FUNCTION_BLOCK "FB303"   // FB303, LAD
TITLE = FB303
{ S7_Optimized_Access := 'TRUE' }
AUTHOR : PRECISE
FAMILY : PRECISE
// SPARGING
// stored: AutoNumber false, MemoryReserve 100, SetENOAutomatically false
   VAR_INPUT
      Enable : Bool;
      Disable : Bool;
      Fault : Bool;
      SecPulse : Bool;
      AlwaysTrue { ExternalVisible := 'False'} : Bool;
      StartConfirmationPopupSel : Bool;   // StartConfirmationPopupSel: 0-NO/1-YES
      EndConfirmationPopupSel : Bool;   // EndConfirmationPopupSel: 0-NO/1-YES
      SpargingModeSel : Int;   // Sparging Mode Selection: 0-DO/1-Time
      SpargingTimebaseSel : Bool;   // Sparging Timebase Selection: 0-sec/1-min
      SpargingLineSel : Bool;   // Sparging LineSelection: 0-THRU GAS FILTER /1-THRU VV
      GasSel : Int;   // Gas Selection - 0-AIR/1-N2
      SetDO : Real := 10.0;   // For Sparging Mode Selection: 0-DO
      SpargingTimeMin : Int := 1;   // For Sparging Mode Selection: 1-Time & Sparging Timebase Selection: 1-min
      SpargingTimeSec : Int := 30;   // For Sparging Mode Selection: 1-Time & Sparging Timebase Selection: 0-sec
      PressuretoOpenVV : Real := 1.0;   // For Sparging LineSelection: 1-THRU VV
      PressuretoCloseVV : Real := 0.5;   // For Sparging LineSelection: 1-THRU VV
      ActualDO : Real;   // For Sparging Mode Selection: 0-DO
      ActualPressure : Real;   // For Sparging LineSelection: 1-THRU VV
      DelaytoOpenGasIn : Int := 3;
   END_VAR
   VAR_OUTPUT
      AirValve : Bool;
      N2Valve : Bool;
      SpargingLineValves : Bool;
      VentValve : Bool;   // For Sparging LineSelection: 1-THRU VV
      StartConfirmationPopup : Bool;   // For Start Confirmation Popup Selection: Yes
      EndConfirmationPopup : Bool;   // For End Confirmation Popup Selection: Yes
      SpargingTimeMinPV : DInt;
      SpargingTimeSecPV : DInt;
      PrintTrigger { ExternalAccessible := 'False'; ExternalVisible := 'False'; ExternalWritable := 'False'} : Bool;
      PrintWord : Int;
      PrintStatus : String[50];
   END_VAR
   VAR_IN_OUT
      Start : Bool;
      Stop : Bool;
      Reset : Bool;
      StartConfirmationAck : Bool;   // For Start Confirmation Popup Selection: Yes
      EndConfirmationAck : Bool;   // For End Confirmation Popup Selection: Yes
      SpareBtn1 : Bool;
      SpareBtn2 : Bool;
      SpareBtn3 : Bool;
      Running : Bool;
      Selected : Bool;
      Paused : Bool;
      StartConfirmationPopupTemp : Bool;   // For Start Confirmation Popup Selection: Yes
      EndConfirmationPopupTemp : Bool;   // For End Confirmation Popup Selection: Yes
      SpargingStarted : Bool;
      SpargingOver : Bool;
      SpargingTimerRunning : Bool;
   END_VAR
   VAR
      ValveOnDelayPV : Int;
      ValveOffDelayPV : Int;
      PrintTriggerTemp : Bool;
      RE1 : Bool;
      RE2 : Bool;
      RE3 : Bool;
      RE4 : Bool;
      RE5 : Bool;
      RE6 : Bool;
      RE7 : Bool;
      SpargingTimer : "FB101";
      PrintTriggerResetTimer { S7_SetPoint := 'True'} : TON_TIME;
      BtnResetTimer { S7_SetPoint := 'True'} : TON_TIME;
   END_VAR
   VAR_TEMP
      STATUS1 : String[40];
      STATUS2 : String[40];
      STATUS3 : String[40];
      STATUS4 : String[40];
      STATUS5 : String[40];
   END_VAR
   VAR_TEMP   // added for the SCL form of the ladder/FBD networks
      _w1 : Bool;
      _w2 : Bool;
      _w3 : Bool;
      _w4 : Bool;
      _w5 : Bool;
   END_VAR
BEGIN

REGION Network 1: Running
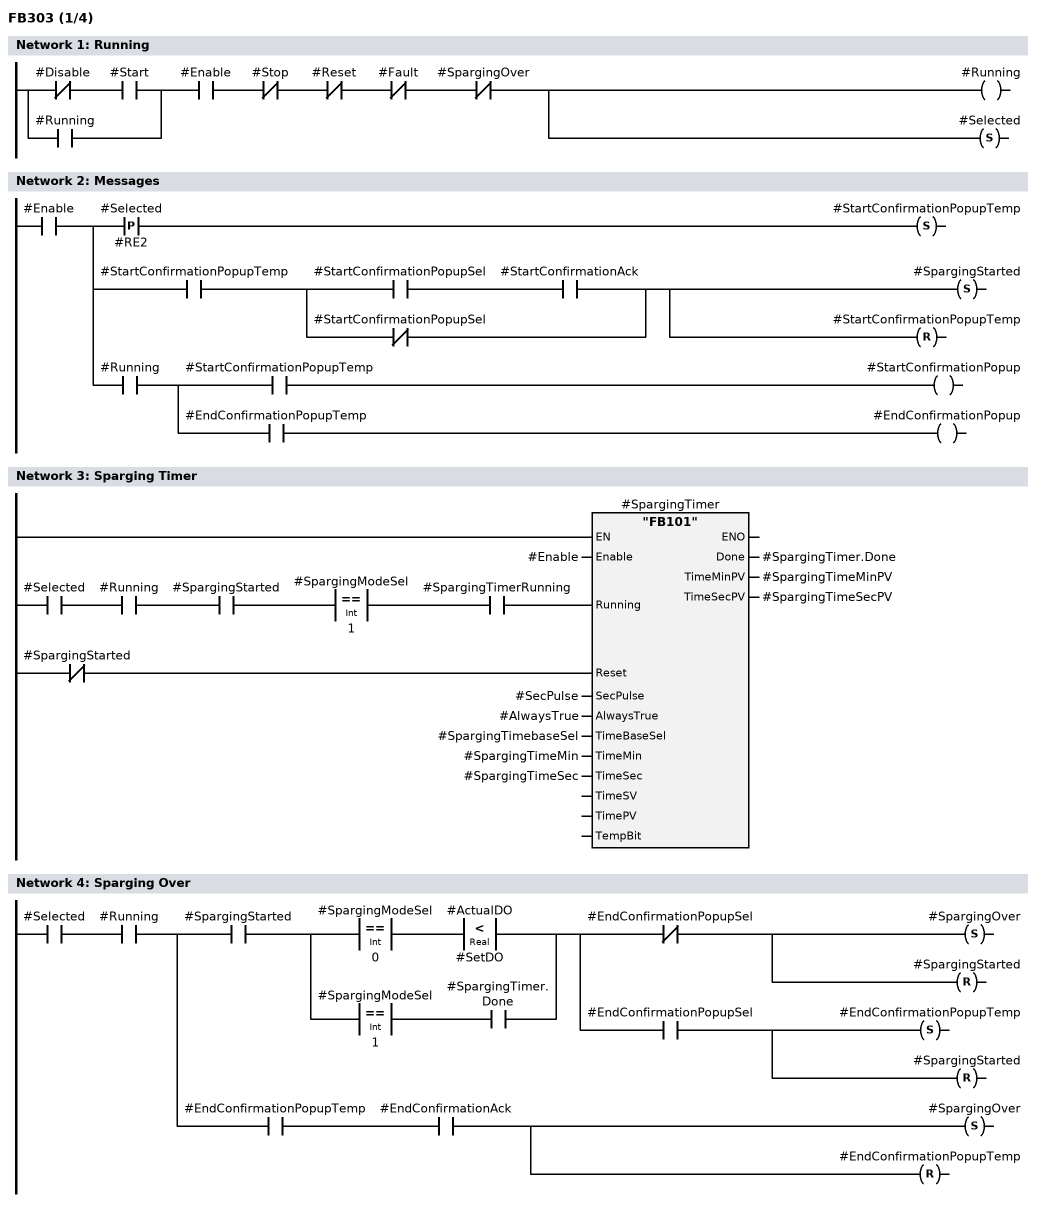
   RUNG wire#powerrail
      I_Contact( #Disable )
      Contact( #Start )
      wire#w1
      Contact( #Enable )
      I_Contact( #Stop )
      I_Contact( #Reset )
      I_Contact( #Fault )
      I_Contact( #SpargingOver )
      wire#w2
      Coil( #Running )
   END_RUNG
   RUNG wire#powerrail
      Contact( #Running )
   END_RUNG wire#w1
   RUNG wire#w2
      S_Coil( #Selected )
   END_RUNG
   // the same network as SCL:
   #Running := ((NOT #Disable AND #Start) OR #Running) AND #Enable AND NOT #Stop AND NOT #Reset AND NOT #Fault AND NOT #SpargingOver;
   IF #Running THEN #Selected := TRUE; END_IF;
END_REGION

REGION Network 2: Messages
   RUNG wire#powerrail
      Contact( #Enable )
      wire#w1
      P_Contact(operand := #Selected, bit := #RE2)
      S_Coil( #StartConfirmationPopupTemp )
   END_RUNG
   RUNG wire#w1
      Contact( #StartConfirmationPopupTemp )
      wire#w2
      Contact( #StartConfirmationPopupSel )
      Contact( #StartConfirmationAck )
      wire#w3
      S_Coil( #SpargingStarted )
   END_RUNG
   RUNG wire#w2
      I_Contact( #StartConfirmationPopupSel )
   END_RUNG wire#w3
   RUNG wire#w3
      R_Coil( #StartConfirmationPopupTemp )
   END_RUNG
   RUNG wire#w1
      Contact( #Running )
      wire#w4
      Contact( #StartConfirmationPopupTemp )
      Coil( #StartConfirmationPopup )
   END_RUNG
   RUNG wire#w4
      Contact( #EndConfirmationPopupTemp )
      Coil( #EndConfirmationPopup )
   END_RUNG
   // the same network as SCL:
   #_w1 := #Enable AND #Selected AND NOT #RE2;   // rising edge of #Selected
   #RE2 := #Selected;
   IF #_w1 THEN #StartConfirmationPopupTemp := TRUE; END_IF;
   IF #Enable AND #StartConfirmationPopupTemp AND ((#StartConfirmationPopupSel AND #StartConfirmationAck) OR NOT #StartConfirmationPopupSel) THEN
       #SpargingStarted := TRUE;
       #StartConfirmationPopupTemp := FALSE;
   END_IF;
   #_w2 := #Enable AND #Running;
   #StartConfirmationPopup := #_w2 AND #StartConfirmationPopupTemp;
   #EndConfirmationPopup := #_w2 AND #EndConfirmationPopupTemp;
END_REGION

REGION Network 3: Sparging Timer
   RUNG wire#powerrail
      #SpargingTimer(Running := wire#w1, Reset := wire#w2, Enable := #Enable, SecPulse := #SecPulse, AlwaysTrue := #AlwaysTrue, TimeBaseSel := #SpargingTimebaseSel, TimeMin := #SpargingTimeMin, TimeSec := #SpargingTimeSec, TimeSV :=, TimePV :=, TempBit :=, Done => #SpargingTimer.Done, TimeMinPV => #SpargingTimeMinPV, TimeSecPV => #SpargingTimeSecPV)
   END_RUNG
   RUNG wire#powerrail
      Contact( #Selected )
      Contact( #Running )
      Contact( #SpargingStarted )
      { S7_Templates := "SrcType := Int" } EQ_Contact(in1 := #SpargingModeSel, in2 := 1)
      Contact( #SpargingTimerRunning )
   END_RUNG wire#w1
   RUNG wire#powerrail
      I_Contact( #SpargingStarted )
   END_RUNG wire#w2
   // the same network as SCL:
   #SpargingTimer(Enable := #Enable,   // "FB101"
                  Running := #Selected AND #Running AND #SpargingStarted AND (#SpargingModeSel = 1) AND #SpargingTimerRunning,
                  Reset := NOT #SpargingStarted,
                  SecPulse := #SecPulse,
                  AlwaysTrue := #AlwaysTrue,
                  TimeBaseSel := #SpargingTimebaseSel,
                  TimeMin := #SpargingTimeMin,
                  TimeSec := #SpargingTimeSec,
                  Done => #SpargingTimer.Done,
                  TimeMinPV => #SpargingTimeMinPV,
                  TimeSecPV => #SpargingTimeSecPV);
END_REGION

REGION Network 4: Sparging Over
   RUNG wire#powerrail
      Contact( #Selected )
      Contact( #Running )
      wire#w1
      Contact( #SpargingStarted )
      wire#w2
      { S7_Templates := "SrcType := Int" } EQ_Contact(in1 := #SpargingModeSel, in2 := 0)
      { S7_Templates := "SrcType := Real" } LT_Contact(in1 := #ActualDO, in2 := #SetDO)
      wire#w3
      I_Contact( #EndConfirmationPopupSel )
      wire#w4
      S_Coil( #SpargingOver )
   END_RUNG
   RUNG wire#w2
      { S7_Templates := "SrcType := Int" } EQ_Contact(in1 := #SpargingModeSel, in2 := 1)
      Contact( #SpargingTimer.Done )
   END_RUNG wire#w3
   RUNG wire#w4
      R_Coil( #SpargingStarted )
   END_RUNG
   RUNG wire#w3
      Contact( #EndConfirmationPopupSel )
      wire#w5
      S_Coil( #EndConfirmationPopupTemp )
   END_RUNG
   RUNG wire#w5
      R_Coil( #SpargingStarted )
   END_RUNG
   RUNG wire#w1
      Contact( #EndConfirmationPopupTemp )
      Contact( #EndConfirmationAck )
      wire#w6
      S_Coil( #SpargingOver )
   END_RUNG
   RUNG wire#w6
      R_Coil( #EndConfirmationPopupTemp )
   END_RUNG
   // the same network as SCL:
   #_w1 := #Selected AND #Running;
   #_w2 := #_w1 AND #SpargingStarted AND (((#SpargingModeSel = 0) AND (#ActualDO < #SetDO)) OR ((#SpargingModeSel = 1) AND #SpargingTimer.Done));
   IF #_w2 AND NOT #EndConfirmationPopupSel THEN
       #SpargingOver := TRUE;
       #SpargingStarted := FALSE;
   END_IF;
   IF #_w2 AND #EndConfirmationPopupSel THEN
       #EndConfirmationPopupTemp := TRUE;
       #SpargingStarted := FALSE;
   END_IF;
   IF #_w1 AND #EndConfirmationPopupTemp AND #EndConfirmationAck THEN
       #SpargingOver := TRUE;
       #EndConfirmationPopupTemp := FALSE;
   END_IF;
END_REGION

REGION Network 5: Output On
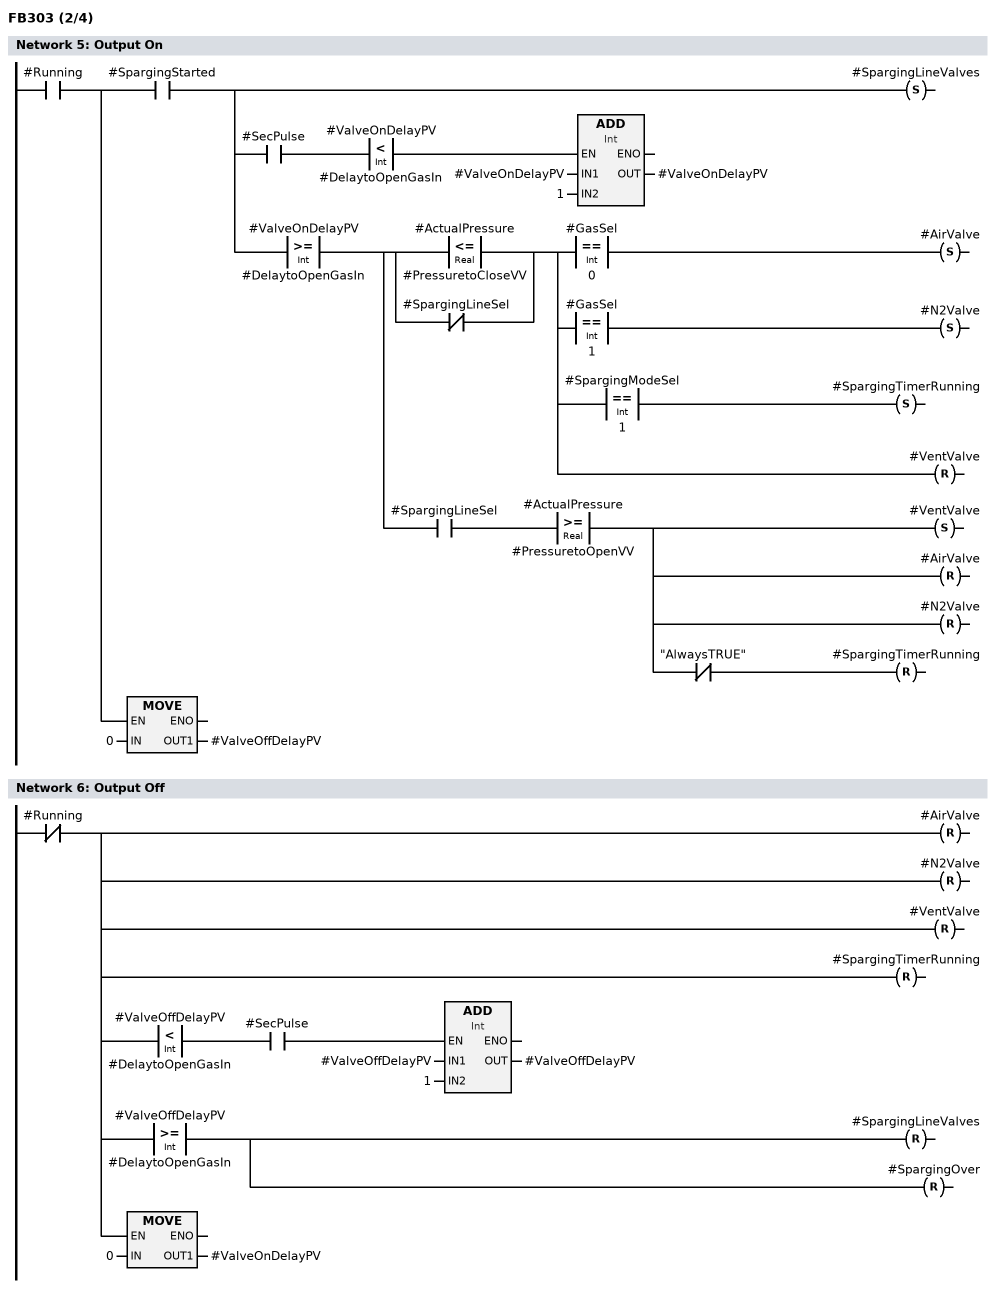
   RUNG wire#powerrail
      Contact( #Running )
      wire#w1
      Contact( #SpargingStarted )
      wire#w2
      S_Coil( #SpargingLineValves )
   END_RUNG
   RUNG wire#w2
      Contact( #SecPulse )
      { S7_Templates := "SrcType := Int" } LT_Contact(in1 := #ValveOnDelayPV, in2 := #DelaytoOpenGasIn)
      { S7_Templates := "SrcType := Int"; S7_GenerateENO := "TRUE" } Add(in1 := #ValveOnDelayPV, in2 := 1, out => #ValveOnDelayPV)
   END_RUNG
   RUNG wire#w2
      { S7_Templates := "SrcType := Int" } GE_Contact(in1 := #ValveOnDelayPV, in2 := #DelaytoOpenGasIn)
      wire#w3
      { S7_Templates := "SrcType := Real" } LE_Contact(in1 := #ActualPressure, in2 := #PressuretoCloseVV)
      wire#w4
      { S7_Templates := "SrcType := Int" } EQ_Contact(in1 := #GasSel, in2 := 0)
      S_Coil( #AirValve )
   END_RUNG
   RUNG wire#w3
      I_Contact( #SpargingLineSel )
   END_RUNG wire#w4
   RUNG wire#w4
      { S7_Templates := "SrcType := Int" } EQ_Contact(in1 := #GasSel, in2 := 1)
      S_Coil( #N2Valve )
   END_RUNG
   RUNG wire#w4
      { S7_Templates := "SrcType := Int" } EQ_Contact(in1 := #SpargingModeSel, in2 := 1)
      S_Coil( #SpargingTimerRunning )
   END_RUNG
   RUNG wire#w4
      R_Coil( #VentValve )
   END_RUNG
   RUNG wire#w3
      Contact( #SpargingLineSel )
      { S7_Templates := "SrcType := Real" } GE_Contact(in1 := #ActualPressure, in2 := #PressuretoOpenVV)
      wire#w5
      S_Coil( #VentValve )
   END_RUNG
   RUNG wire#w5
      R_Coil( #AirValve )
   END_RUNG
   RUNG wire#w5
      R_Coil( #N2Valve )
   END_RUNG
   RUNG wire#w5
      I_Contact( "AlwaysTRUE" )
      R_Coil( #SpargingTimerRunning )
   END_RUNG
   RUNG wire#w1
      { S7_GenerateENO := "TRUE" } Move(in := 0, out1 => #ValveOffDelayPV)
   END_RUNG
   // the same network as SCL:
   #_w1 := #Running AND #SpargingStarted;
   IF #_w1 THEN #SpargingLineValves := TRUE; END_IF;
   IF #_w1 AND #SecPulse AND (#ValveOnDelayPV < #DelaytoOpenGasIn) THEN
       #ValveOnDelayPV := #ValveOnDelayPV + 1;
   END_IF;
   #_w2 := #_w1 AND (#ValveOnDelayPV >= #DelaytoOpenGasIn);
   #_w3 := #_w2 AND ((#ActualPressure <= #PressuretoCloseVV) OR NOT #SpargingLineSel);
   IF #_w3 AND (#GasSel = 0) THEN #AirValve := TRUE; END_IF;
   IF #_w3 AND (#GasSel = 1) THEN #N2Valve := TRUE; END_IF;
   IF #_w3 AND (#SpargingModeSel = 1) THEN #SpargingTimerRunning := TRUE; END_IF;
   IF #_w3 THEN #VentValve := FALSE; END_IF;
   #_w4 := #_w2 AND #SpargingLineSel AND (#ActualPressure >= #PressuretoOpenVV);
   IF #_w4 THEN
       #VentValve := TRUE;
       #AirValve := FALSE;
       #N2Valve := FALSE;
   END_IF;
   IF #_w4 AND NOT "AlwaysTRUE" THEN #SpargingTimerRunning := FALSE; END_IF;
   IF #Running THEN #ValveOffDelayPV := 0; END_IF;
END_REGION

REGION Network 6: Output Off
   RUNG wire#powerrail
      I_Contact( #Running )
      wire#w1
      R_Coil( #AirValve )
   END_RUNG
   RUNG wire#w1
      R_Coil( #N2Valve )
   END_RUNG
   RUNG wire#w1
      R_Coil( #VentValve )
   END_RUNG
   RUNG wire#w1
      R_Coil( #SpargingTimerRunning )
   END_RUNG
   RUNG wire#w1
      { S7_Templates := "SrcType := Int" } LT_Contact(in1 := #ValveOffDelayPV, in2 := #DelaytoOpenGasIn)
      Contact( #SecPulse )
      { S7_Templates := "SrcType := Int"; S7_GenerateENO := "TRUE" } Add(in1 := #ValveOffDelayPV, in2 := 1, out => #ValveOffDelayPV)
   END_RUNG
   RUNG wire#w1
      { S7_Templates := "SrcType := Int" } GE_Contact(in1 := #ValveOffDelayPV, in2 := #DelaytoOpenGasIn)
      wire#w2
      R_Coil( #SpargingLineValves )
   END_RUNG
   RUNG wire#w2
      R_Coil( #SpargingOver )
   END_RUNG
   RUNG wire#w1
      { S7_GenerateENO := "TRUE" } Move(in := 0, out1 => #ValveOnDelayPV)
   END_RUNG
   // the same network as SCL:
   IF NOT #Running THEN
       #AirValve := FALSE;
       #N2Valve := FALSE;
       #VentValve := FALSE;
       #SpargingTimerRunning := FALSE;
   END_IF;
   IF NOT #Running AND (#ValveOffDelayPV < #DelaytoOpenGasIn) AND #SecPulse THEN
       #ValveOffDelayPV := #ValveOffDelayPV + 1;
   END_IF;
   IF NOT #Running AND (#ValveOffDelayPV >= #DelaytoOpenGasIn) THEN
       #SpargingLineValves := FALSE;
       #SpargingOver := FALSE;
   END_IF;
   IF NOT #Running THEN #ValveOnDelayPV := 0; END_IF;
END_REGION

REGION Network 7: Event Status
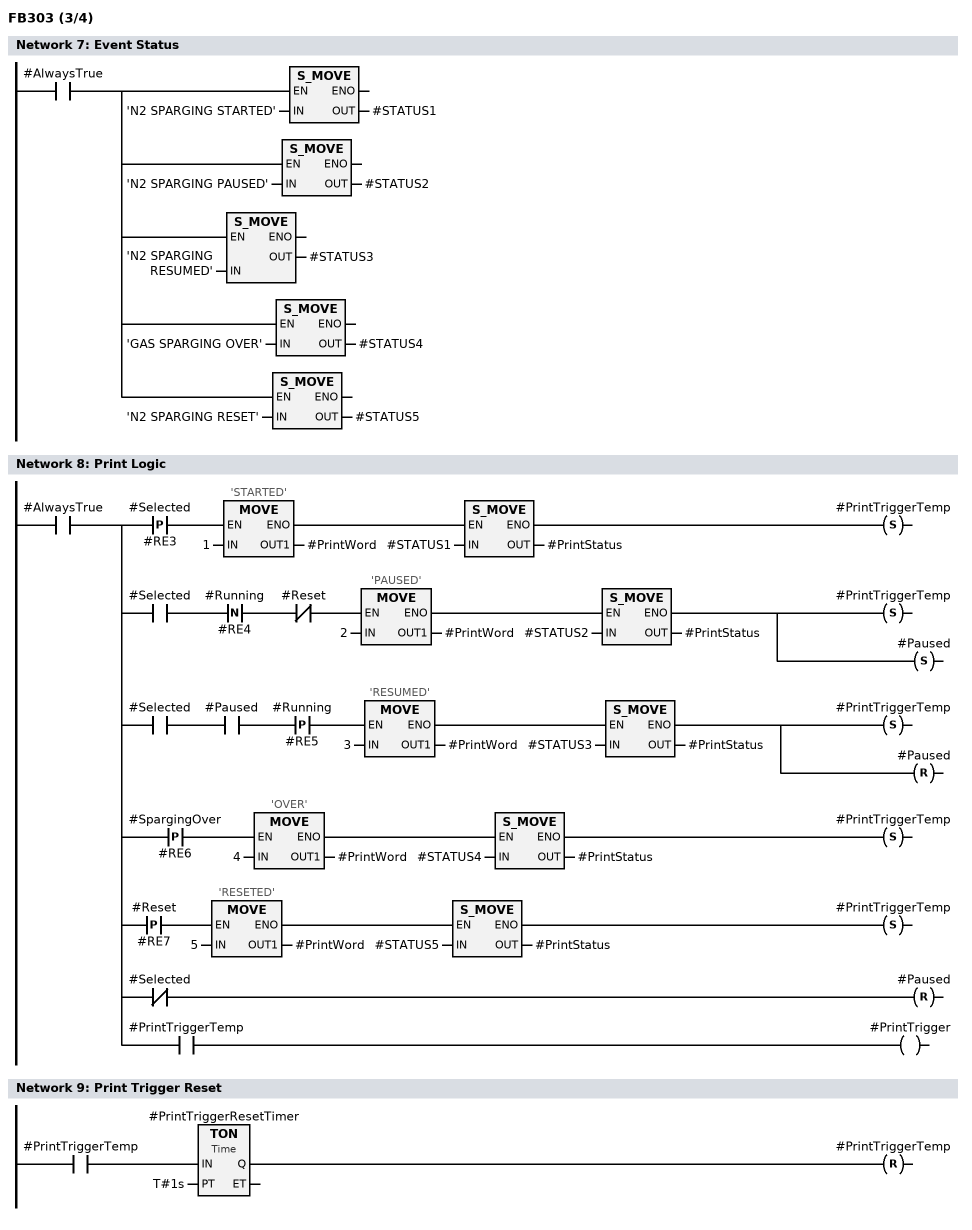
   RUNG wire#powerrail
      Contact( #AlwaysTrue )
      wire#w1
      S_Move(in := 'N2 SPARGING STARTED', out => #STATUS1)
   END_RUNG
   RUNG wire#w1
      S_Move(in := 'N2 SPARGING PAUSED', out => #STATUS2)
   END_RUNG
   RUNG wire#w1
      S_Move(in := 'N2 SPARGING RESUMED', out => #STATUS3)
   END_RUNG
   RUNG wire#w1
      S_Move(in := 'GAS SPARGING OVER', out => #STATUS4)
   END_RUNG
   RUNG wire#w1
      S_Move(in := 'N2 SPARGING RESET', out => #STATUS5)
   END_RUNG
   // the same network as SCL:
   IF #AlwaysTrue THEN
       #STATUS1 := 'N2 SPARGING STARTED';
       #STATUS2 := 'N2 SPARGING PAUSED';
       #STATUS3 := 'N2 SPARGING RESUMED';
       #STATUS4 := 'GAS SPARGING OVER';
       #STATUS5 := 'N2 SPARGING RESET';
   END_IF;
END_REGION

REGION Network 8: Print Logic
   RUNG wire#powerrail
      Contact( #AlwaysTrue )
      wire#w1
      P_Contact(operand := #Selected, bit := #RE3)
      { S7_GenerateENO := "TRUE" } Move(in := 1, out1 => #PrintWord)   // 'STARTED'
      S_Move(in := #STATUS1, out => #PrintStatus)
      S_Coil( #PrintTriggerTemp )
   END_RUNG
   RUNG wire#w1
      Contact( #Selected )
      N_Contact(operand := #Running, bit := #RE4)
      I_Contact( #Reset )
      { S7_GenerateENO := "TRUE" } Move(in := 2, out1 => #PrintWord)   // 'PAUSED'
      S_Move(in := #STATUS2, out => #PrintStatus)
      wire#w2
      S_Coil( #PrintTriggerTemp )
   END_RUNG
   RUNG wire#w2
      S_Coil( #Paused )
   END_RUNG
   RUNG wire#w1
      Contact( #Selected )
      Contact( #Paused )
      P_Contact(operand := #Running, bit := #RE5)
      { S7_GenerateENO := "TRUE" } Move(in := 3, out1 => #PrintWord)   // 'RESUMED'
      S_Move(in := #STATUS3, out => #PrintStatus)
      wire#w3
      S_Coil( #PrintTriggerTemp )
   END_RUNG
   RUNG wire#w3
      R_Coil( #Paused )
   END_RUNG
   RUNG wire#w1
      P_Contact(operand := #SpargingOver, bit := #RE6)
      { S7_GenerateENO := "TRUE" } Move(in := 4, out1 => #PrintWord)   // 'OVER'
      S_Move(in := #STATUS4, out => #PrintStatus)
      S_Coil( #PrintTriggerTemp )
   END_RUNG
   RUNG wire#w1
      P_Contact(operand := #Reset, bit := #RE7)
      { S7_GenerateENO := "TRUE" } Move(in := 5, out1 => #PrintWord)   // 'RESETED'
      S_Move(in := #STATUS5, out => #PrintStatus)
      S_Coil( #PrintTriggerTemp )
   END_RUNG
   RUNG wire#w1
      I_Contact( #Selected )
      R_Coil( #Paused )
   END_RUNG
   RUNG wire#w1
      Contact( #PrintTriggerTemp )
      Coil( #PrintTrigger )
   END_RUNG
   // the same network as SCL:
   // ENO of a box is taken as its EN; it also drops when the box reports an error
   #_w1 := #AlwaysTrue AND #Selected AND NOT #RE3;   // rising edge of #Selected
   #RE3 := #Selected;
   IF #_w1 THEN
       #PrintWord := 1;   // 'STARTED'
       #PrintStatus := #STATUS1;
       #PrintTriggerTemp := TRUE;
   END_IF;
   #_w2 := #AlwaysTrue AND #Selected AND NOT #Running AND #RE4;   // falling edge of #Running
   #RE4 := #Running;
   IF #_w2 AND NOT #Reset THEN
       #PrintWord := 2;   // 'PAUSED'
       #PrintStatus := #STATUS2;
       #PrintTriggerTemp := TRUE;
       #Paused := TRUE;
   END_IF;
   #_w3 := #AlwaysTrue AND #Selected AND #Paused AND #Running AND NOT #RE5;   // rising edge of #Running
   #RE5 := #Running;
   IF #_w3 THEN
       #PrintWord := 3;   // 'RESUMED'
       #PrintStatus := #STATUS3;
       #PrintTriggerTemp := TRUE;
       #Paused := FALSE;
   END_IF;
   #_w4 := #AlwaysTrue AND #SpargingOver AND NOT #RE6;   // rising edge of #SpargingOver
   #RE6 := #SpargingOver;
   IF #_w4 THEN
       #PrintWord := 4;   // 'OVER'
       #PrintStatus := #STATUS4;
       #PrintTriggerTemp := TRUE;
   END_IF;
   #_w5 := #AlwaysTrue AND #Reset AND NOT #RE7;   // rising edge of #Reset
   #RE7 := #Reset;
   IF #_w5 THEN
       #PrintWord := 5;   // 'RESETED'
       #PrintStatus := #STATUS5;
       #PrintTriggerTemp := TRUE;
   END_IF;
   IF #AlwaysTrue AND NOT #Selected THEN #Paused := FALSE; END_IF;
   #PrintTrigger := #AlwaysTrue AND #PrintTriggerTemp;
END_REGION

REGION Network 9: Print Trigger Reset
   RUNG wire#powerrail
      Contact( #PrintTriggerTemp )
      { S7_Templates := "time_type := Time" } #PrintTriggerResetTimer.TON(pt := T#1s, et =>)
      R_Coil( #PrintTriggerTemp )
   END_RUNG
   // the same network as SCL:
   #PrintTriggerResetTimer(IN := #PrintTriggerTemp, PT := T#1s);   // TON
   IF #PrintTriggerResetTimer.Q THEN #PrintTriggerTemp := FALSE; END_IF;
END_REGION

REGION Network 10: Button Reset
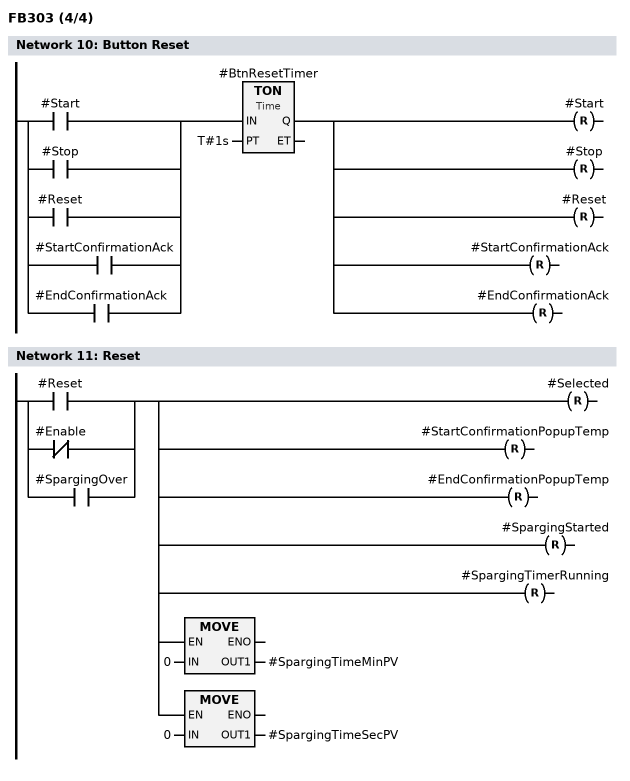
   RUNG wire#powerrail
      Contact( #Start )
      wire#w1
      { S7_Templates := "time_type := Time" } #BtnResetTimer.TON(pt := T#1s, et =>)
      wire#w2
      R_Coil( #Start )
   END_RUNG
   RUNG wire#powerrail
      Contact( #Stop )
   END_RUNG wire#w1
   RUNG wire#powerrail
      Contact( #Reset )
   END_RUNG wire#w1
   RUNG wire#powerrail
      Contact( #StartConfirmationAck )
   END_RUNG wire#w1
   RUNG wire#powerrail
      Contact( #EndConfirmationAck )
   END_RUNG wire#w1
   RUNG wire#w2
      R_Coil( #Stop )
   END_RUNG
   RUNG wire#w2
      R_Coil( #Reset )
   END_RUNG
   RUNG wire#w2
      R_Coil( #StartConfirmationAck )
   END_RUNG
   RUNG wire#w2
      R_Coil( #EndConfirmationAck )
   END_RUNG
   // the same network as SCL:
   #BtnResetTimer(IN := #Start OR #Stop OR #Reset OR #StartConfirmationAck OR #EndConfirmationAck, PT := T#1s);   // TON
   IF #BtnResetTimer.Q THEN
       #Start := FALSE;
       #Stop := FALSE;
       #Reset := FALSE;
       #StartConfirmationAck := FALSE;
       #EndConfirmationAck := FALSE;
   END_IF;
END_REGION

REGION Network 11: Reset
   RUNG wire#powerrail
      Contact( #Reset )
      wire#w1
      R_Coil( #Selected )
   END_RUNG
   RUNG wire#powerrail
      I_Contact( #Enable )
   END_RUNG wire#w1
   RUNG wire#powerrail
      Contact( #SpargingOver )
   END_RUNG wire#w1
   RUNG wire#w1
      R_Coil( #StartConfirmationPopupTemp )
   END_RUNG
   RUNG wire#w1
      R_Coil( #EndConfirmationPopupTemp )
   END_RUNG
   RUNG wire#w1
      R_Coil( #SpargingStarted )
   END_RUNG
   RUNG wire#w1
      R_Coil( #SpargingTimerRunning )
   END_RUNG
   RUNG wire#w1
      { S7_GenerateENO := "TRUE" } Move(in := 0, out1 => #SpargingTimeMinPV)
   END_RUNG
   RUNG wire#w1
      { S7_GenerateENO := "TRUE" } Move(in := 0, out1 => #SpargingTimeSecPV)
   END_RUNG
   // the same network as SCL:
   IF #Reset OR NOT #Enable OR #SpargingOver THEN
       #Selected := FALSE;
       #StartConfirmationPopupTemp := FALSE;
       #EndConfirmationPopupTemp := FALSE;
       #SpargingStarted := FALSE;
       #SpargingTimerRunning := FALSE;
       #SpargingTimeMinPV := 0;
       #SpargingTimeSecPV := 0;
   END_IF;
END_REGION
END_FUNCTION_BLOCK

FUNCTION_BLOCK "FB304"   // FB304, LAD
TITLE = FB304
{ S7_Optimized_Access := 'TRUE' }
AUTHOR : PRECISE
FAMILY : PRECISE
// BLANKETING
// stored: AutoNumber false, MemoryReserve 100, SetENOAutomatically false
   VAR_INPUT
      Enable : Bool;
      Disable : Bool;
      Fault : Bool;
      SecPulse : Bool;
      AlwaysTrue : Bool;
      StartConfirmationPopupSel : Bool;   // StartConfirmationPopupSel: 0-NO/1-YES
      EndConfirmationPopupSel : Bool;   // EndConfirmationPopupSel: 0-NO/1-YES
      BlanketingModeSel : Int;   // Blanketing Mode Selection: 0-Pressure/1-Pressure+Time
      BlanketingTimebaseSel : Bool;   // Blanketing Timebase Selection: 0-sec/1-min
      GasSel : Int;   // Gas Selection - 0-AIR/1-N2
      SetPressure : Real := 1.0;   // For Blanketing Mode Selection: 0-Pressure
      BlanketingTimeMin : Int := 1;   // For Blanketing Mode Selection: 1-Pressure+Time & Blanketing Timebase Selection: 1-min
      BlanketingTimeSec : Int := 30;   // For Blanketing Mode Selection: 1-Pressure+Time & Blanketing Timebase Selection: 0-sec
      ActualPressure : Real;   // For Sparging LineSelection: 1-THRU VV
      DelaytoOpenGasIn : Int := 3;
      PressureTol : Real := 0.3;
   END_VAR
   VAR_OUTPUT
      AirValve : Bool;
      N2Valve : Bool;
      BlanketingLineValves : Bool;
      StartConfirmationPopup : Bool;   // For Start Confirmation Popup Selection: Yes
      EndConfirmationPopup : Bool;   // For End Confirmation Popup Selection: Yes
      BlanketingTimeMinPV : DInt;
      BlanketingTimeSecPV : DInt;
      PrintTrigger : Bool;
      PrintWord : Int;
      PrintStatus : String[50];
   END_VAR
   VAR_IN_OUT
      Start : Bool;
      Stop : Bool;
      Reset : Bool;
      StartConfirmationAck : Bool;   // For Start Confirmation Popup Selection: Yes
      EndConfirmationAck : Bool;   // For End Confirmation Popup Selection: Yes
      SpareBtn1 : Bool;
      SpareBtn2 : Bool;
      SpareBtn3 : Bool;
      Running : Bool;
      Selected : Bool;
      Paused : Bool;
      StartConfirmationPopupTemp : Bool;   // For Start Confirmation Popup Selection: Yes
      EndConfirmationPopupTemp : Bool;   // For End Confirmation Popup Selection: Yes
      BlanketingStarted : Bool;
      BlanketingOver : Bool;
      BlanketingTimerRunning : Bool;
      PressureTolNeg : Real;
   END_VAR
   VAR
      ValveOnDelayPV : Int;
      ValveOffDelayPV : Int;
      PrintTriggerTemp : Bool;
      RE1 : Bool;
      RE2 : Bool;
      RE3 : Bool;
      RE4 : Bool;
      RE5 : Bool;
      RE6 : Bool;
      RE7 : Bool;
      BlanketingTimer { S7_SetPoint := 'True'} : "FB101";
      PrintTriggerResetTimer { S7_SetPoint := 'True'} : TON_TIME;
      BtnResetTimer { S7_SetPoint := 'True'} : TON_TIME;
   END_VAR
   VAR_TEMP
      STATUS1 : String[40];
      STATUS2 : String[40];
      STATUS3 : String[40];
      STATUS4 : String[40];
      STATUS5 : String[40];
   END_VAR
   VAR_TEMP   // added for the SCL form of the ladder/FBD networks
      _w1 : Bool;
      _w2 : Bool;
      _w3 : Bool;
      _w4 : Bool;
      _w5 : Bool;
   END_VAR
BEGIN

REGION Network 1: Running
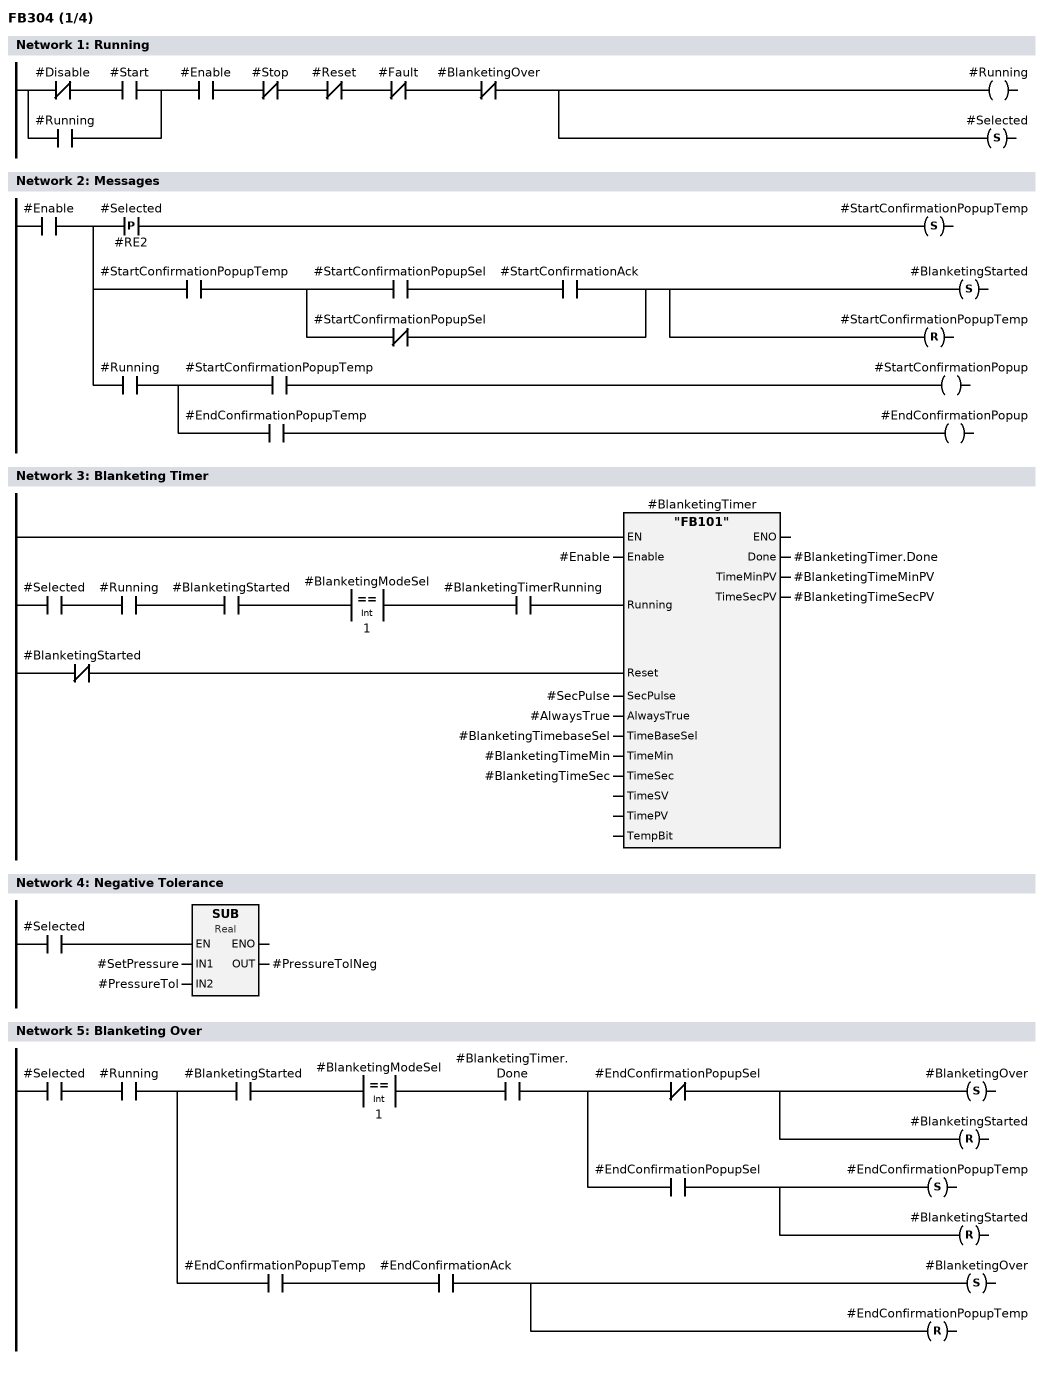
   RUNG wire#powerrail
      I_Contact( #Disable )
      Contact( #Start )
      wire#w1
      Contact( #Enable )
      I_Contact( #Stop )
      I_Contact( #Reset )
      I_Contact( #Fault )
      I_Contact( #BlanketingOver )
      wire#w2
      Coil( #Running )
   END_RUNG
   RUNG wire#powerrail
      Contact( #Running )
   END_RUNG wire#w1
   RUNG wire#w2
      S_Coil( #Selected )
   END_RUNG
   // the same network as SCL:
   #Running := ((NOT #Disable AND #Start) OR #Running) AND #Enable AND NOT #Stop AND NOT #Reset AND NOT #Fault AND NOT #BlanketingOver;
   IF #Running THEN #Selected := TRUE; END_IF;
END_REGION

REGION Network 2: Messages
   RUNG wire#powerrail
      Contact( #Enable )
      wire#w1
      P_Contact(operand := #Selected, bit := #RE2)
      S_Coil( #StartConfirmationPopupTemp )
   END_RUNG
   RUNG wire#w1
      Contact( #StartConfirmationPopupTemp )
      wire#w2
      Contact( #StartConfirmationPopupSel )
      Contact( #StartConfirmationAck )
      wire#w3
      S_Coil( #BlanketingStarted )
   END_RUNG
   RUNG wire#w2
      I_Contact( #StartConfirmationPopupSel )
   END_RUNG wire#w3
   RUNG wire#w3
      R_Coil( #StartConfirmationPopupTemp )
   END_RUNG
   RUNG wire#w1
      Contact( #Running )
      wire#w4
      Contact( #StartConfirmationPopupTemp )
      Coil( #StartConfirmationPopup )
   END_RUNG
   RUNG wire#w4
      Contact( #EndConfirmationPopupTemp )
      Coil( #EndConfirmationPopup )
   END_RUNG
   // the same network as SCL:
   #_w1 := #Enable AND #Selected AND NOT #RE2;   // rising edge of #Selected
   #RE2 := #Selected;
   IF #_w1 THEN #StartConfirmationPopupTemp := TRUE; END_IF;
   IF #Enable AND #StartConfirmationPopupTemp AND ((#StartConfirmationPopupSel AND #StartConfirmationAck) OR NOT #StartConfirmationPopupSel) THEN
       #BlanketingStarted := TRUE;
       #StartConfirmationPopupTemp := FALSE;
   END_IF;
   #_w2 := #Enable AND #Running;
   #StartConfirmationPopup := #_w2 AND #StartConfirmationPopupTemp;
   #EndConfirmationPopup := #_w2 AND #EndConfirmationPopupTemp;
END_REGION

REGION Network 3: Blanketing Timer
   RUNG wire#powerrail
      #BlanketingTimer(Running := wire#w1, Reset := wire#w2, Enable := #Enable, SecPulse := #SecPulse, AlwaysTrue := #AlwaysTrue, TimeBaseSel := #BlanketingTimebaseSel, TimeMin := #BlanketingTimeMin, TimeSec := #BlanketingTimeSec, TimeSV :=, TimePV :=, TempBit :=, Done => #BlanketingTimer.Done, TimeMinPV => #BlanketingTimeMinPV, TimeSecPV => #BlanketingTimeSecPV)
   END_RUNG
   RUNG wire#powerrail
      Contact( #Selected )
      Contact( #Running )
      Contact( #BlanketingStarted )
      { S7_Templates := "SrcType := Int" } EQ_Contact(in1 := #BlanketingModeSel, in2 := 1)
      Contact( #BlanketingTimerRunning )
   END_RUNG wire#w1
   RUNG wire#powerrail
      I_Contact( #BlanketingStarted )
   END_RUNG wire#w2
   // the same network as SCL:
   #BlanketingTimer(Enable := #Enable,   // "FB101"
                    Running := #Selected AND #Running AND #BlanketingStarted AND (#BlanketingModeSel = 1) AND #BlanketingTimerRunning,
                    Reset := NOT #BlanketingStarted,
                    SecPulse := #SecPulse,
                    AlwaysTrue := #AlwaysTrue,
                    TimeBaseSel := #BlanketingTimebaseSel,
                    TimeMin := #BlanketingTimeMin,
                    TimeSec := #BlanketingTimeSec,
                    Done => #BlanketingTimer.Done,
                    TimeMinPV => #BlanketingTimeMinPV,
                    TimeSecPV => #BlanketingTimeSecPV);
END_REGION

REGION Network 4: Negative Tolerance
   RUNG wire#powerrail
      Contact( #Selected )
      { S7_Templates := "SrcType := Real"; S7_GenerateENO := "TRUE" } Sub(in1 := #SetPressure, in2 := #PressureTol, out => #PressureTolNeg)
   END_RUNG
   // the same network as SCL:
   IF #Selected THEN #PressureTolNeg := #SetPressure - #PressureTol; END_IF;
END_REGION

REGION Network 5: Blanketing Over
   RUNG wire#powerrail
      Contact( #Selected )
      Contact( #Running )
      wire#w1
      Contact( #BlanketingStarted )
      { S7_Templates := "SrcType := Int" } EQ_Contact(in1 := #BlanketingModeSel, in2 := 1)
      Contact( #BlanketingTimer.Done )
      wire#w2
      I_Contact( #EndConfirmationPopupSel )
      wire#w3
      S_Coil( #BlanketingOver )
   END_RUNG
   RUNG wire#w3
      R_Coil( #BlanketingStarted )
   END_RUNG
   RUNG wire#w2
      Contact( #EndConfirmationPopupSel )
      wire#w4
      S_Coil( #EndConfirmationPopupTemp )
   END_RUNG
   RUNG wire#w4
      R_Coil( #BlanketingStarted )
   END_RUNG
   RUNG wire#w1
      Contact( #EndConfirmationPopupTemp )
      Contact( #EndConfirmationAck )
      wire#w5
      S_Coil( #BlanketingOver )
   END_RUNG
   RUNG wire#w5
      R_Coil( #EndConfirmationPopupTemp )
   END_RUNG
   // the same network as SCL:
   #_w1 := #Selected AND #Running;
   #_w2 := #_w1 AND #BlanketingStarted AND (#BlanketingModeSel = 1) AND #BlanketingTimer.Done;
   IF #_w2 AND NOT #EndConfirmationPopupSel THEN
       #BlanketingOver := TRUE;
       #BlanketingStarted := FALSE;
   END_IF;
   IF #_w2 AND #EndConfirmationPopupSel THEN
       #EndConfirmationPopupTemp := TRUE;
       #BlanketingStarted := FALSE;
   END_IF;
   IF #_w1 AND #EndConfirmationPopupTemp AND #EndConfirmationAck THEN
       #BlanketingOver := TRUE;
       #EndConfirmationPopupTemp := FALSE;
   END_IF;
END_REGION

REGION Network 6: Output On
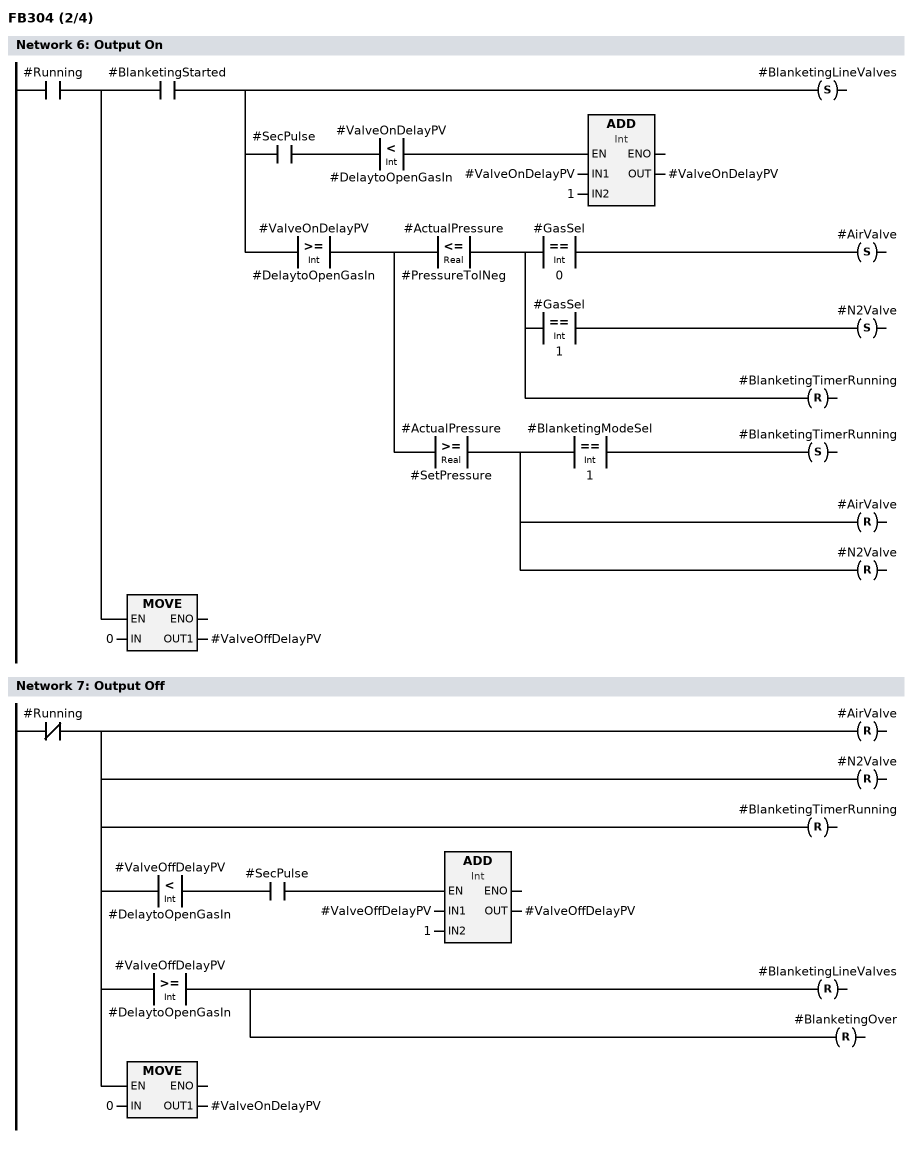
   RUNG wire#powerrail
      Contact( #Running )
      wire#w1
      Contact( #BlanketingStarted )
      wire#w2
      S_Coil( #BlanketingLineValves )
   END_RUNG
   RUNG wire#w2
      Contact( #SecPulse )
      { S7_Templates := "SrcType := Int" } LT_Contact(in1 := #ValveOnDelayPV, in2 := #DelaytoOpenGasIn)
      { S7_Templates := "SrcType := Int"; S7_GenerateENO := "TRUE" } Add(in1 := #ValveOnDelayPV, in2 := 1, out => #ValveOnDelayPV)
   END_RUNG
   RUNG wire#w2
      { S7_Templates := "SrcType := Int" } GE_Contact(in1 := #ValveOnDelayPV, in2 := #DelaytoOpenGasIn)
      wire#w3
      { S7_Templates := "SrcType := Real" } LE_Contact(in1 := #ActualPressure, in2 := #PressureTolNeg)
      wire#w4
      { S7_Templates := "SrcType := Int" } EQ_Contact(in1 := #GasSel, in2 := 0)
      S_Coil( #AirValve )
   END_RUNG
   RUNG wire#w4
      { S7_Templates := "SrcType := Int" } EQ_Contact(in1 := #GasSel, in2 := 1)
      S_Coil( #N2Valve )
   END_RUNG
   RUNG wire#w4
      R_Coil( #BlanketingTimerRunning )
   END_RUNG
   RUNG wire#w3
      { S7_Templates := "SrcType := Real" } GE_Contact(in1 := #ActualPressure, in2 := #SetPressure)
      wire#w5
      { S7_Templates := "SrcType := Int" } EQ_Contact(in1 := #BlanketingModeSel, in2 := 1)
      S_Coil( #BlanketingTimerRunning )
   END_RUNG
   RUNG wire#w5
      R_Coil( #AirValve )
   END_RUNG
   RUNG wire#w5
      R_Coil( #N2Valve )
   END_RUNG
   RUNG wire#w1
      { S7_GenerateENO := "TRUE" } Move(in := 0, out1 => #ValveOffDelayPV)
   END_RUNG
   // the same network as SCL:
   #_w1 := #Running AND #BlanketingStarted;
   IF #_w1 THEN #BlanketingLineValves := TRUE; END_IF;
   IF #_w1 AND #SecPulse AND (#ValveOnDelayPV < #DelaytoOpenGasIn) THEN
       #ValveOnDelayPV := #ValveOnDelayPV + 1;
   END_IF;
   #_w2 := #_w1 AND (#ValveOnDelayPV >= #DelaytoOpenGasIn);
   #_w3 := #_w2 AND (#ActualPressure <= #PressureTolNeg);
   IF #_w3 AND (#GasSel = 0) THEN #AirValve := TRUE; END_IF;
   IF #_w3 AND (#GasSel = 1) THEN #N2Valve := TRUE; END_IF;
   IF #_w3 THEN #BlanketingTimerRunning := FALSE; END_IF;
   #_w4 := #_w2 AND (#ActualPressure >= #SetPressure);
   IF #_w4 AND (#BlanketingModeSel = 1) THEN #BlanketingTimerRunning := TRUE; END_IF;
   IF #_w4 THEN
       #AirValve := FALSE;
       #N2Valve := FALSE;
   END_IF;
   IF #Running THEN #ValveOffDelayPV := 0; END_IF;
END_REGION

REGION Network 7: Output Off
   RUNG wire#powerrail
      I_Contact( #Running )
      wire#w1
      R_Coil( #AirValve )
   END_RUNG
   RUNG wire#w1
      R_Coil( #N2Valve )
   END_RUNG
   RUNG wire#w1
      R_Coil( #BlanketingTimerRunning )
   END_RUNG
   RUNG wire#w1
      { S7_Templates := "SrcType := Int" } LT_Contact(in1 := #ValveOffDelayPV, in2 := #DelaytoOpenGasIn)
      Contact( #SecPulse )
      { S7_Templates := "SrcType := Int"; S7_GenerateENO := "TRUE" } Add(in1 := #ValveOffDelayPV, in2 := 1, out => #ValveOffDelayPV)
   END_RUNG
   RUNG wire#w1
      { S7_Templates := "SrcType := Int" } GE_Contact(in1 := #ValveOffDelayPV, in2 := #DelaytoOpenGasIn)
      wire#w2
      R_Coil( #BlanketingLineValves )
   END_RUNG
   RUNG wire#w2
      R_Coil( #BlanketingOver )
   END_RUNG
   RUNG wire#w1
      { S7_GenerateENO := "TRUE" } Move(in := 0, out1 => #ValveOnDelayPV)
   END_RUNG
   // the same network as SCL:
   IF NOT #Running THEN
       #AirValve := FALSE;
       #N2Valve := FALSE;
       #BlanketingTimerRunning := FALSE;
   END_IF;
   IF NOT #Running AND (#ValveOffDelayPV < #DelaytoOpenGasIn) AND #SecPulse THEN
       #ValveOffDelayPV := #ValveOffDelayPV + 1;
   END_IF;
   IF NOT #Running AND (#ValveOffDelayPV >= #DelaytoOpenGasIn) THEN
       #BlanketingLineValves := FALSE;
       #BlanketingOver := FALSE;
   END_IF;
   IF NOT #Running THEN #ValveOnDelayPV := 0; END_IF;
END_REGION

REGION Network 8: Event Status
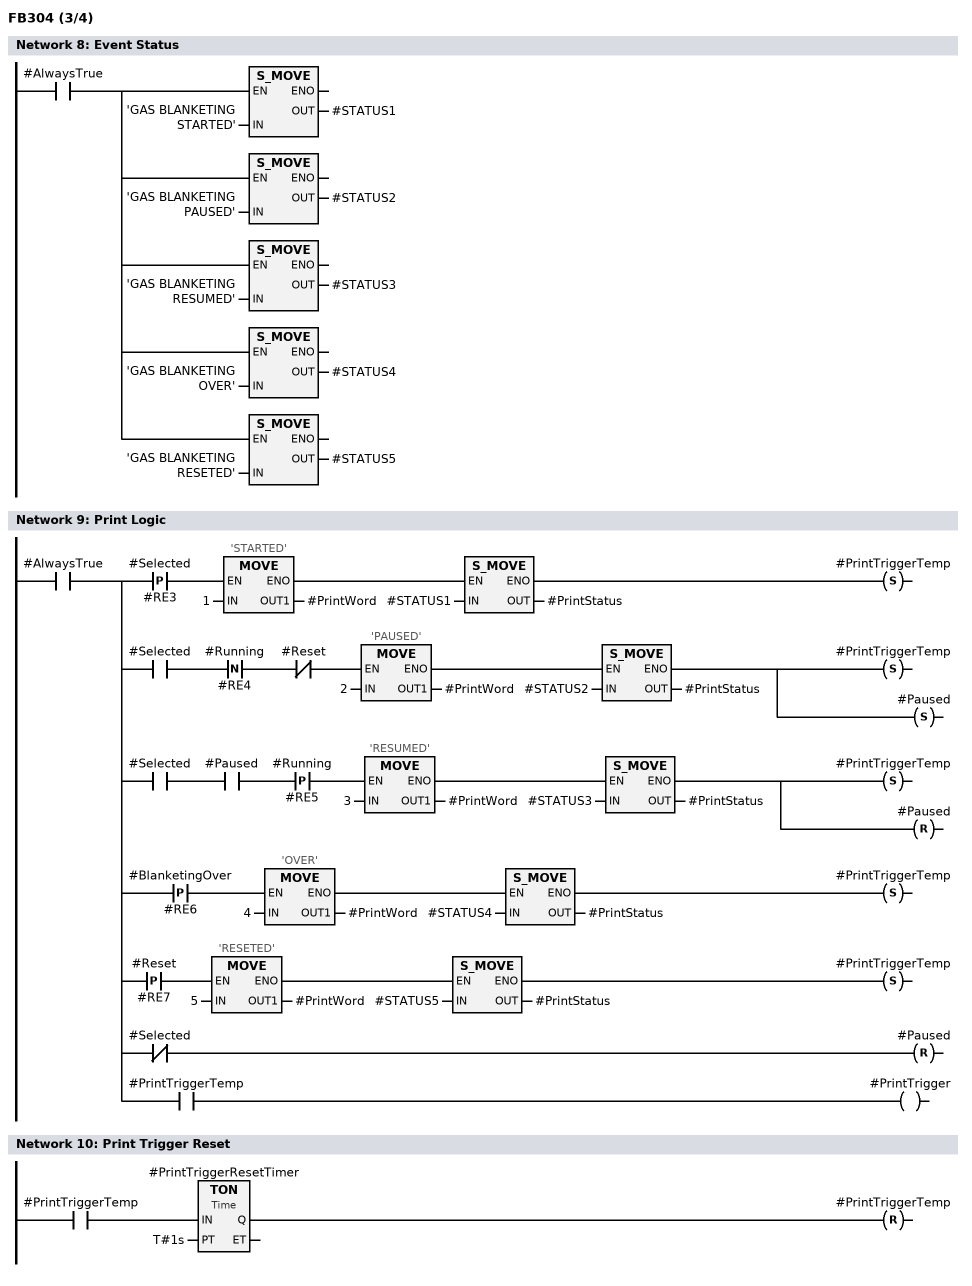
   RUNG wire#powerrail
      Contact( #AlwaysTrue )
      wire#w1
      S_Move(in := 'GAS BLANKETING STARTED', out => #STATUS1)
   END_RUNG
   RUNG wire#w1
      S_Move(in := 'GAS BLANKETING PAUSED', out => #STATUS2)
   END_RUNG
   RUNG wire#w1
      S_Move(in := 'GAS BLANKETING RESUMED', out => #STATUS3)
   END_RUNG
   RUNG wire#w1
      S_Move(in := 'GAS BLANKETING OVER', out => #STATUS4)
   END_RUNG
   RUNG wire#w1
      S_Move(in := 'GAS BLANKETING RESETED', out => #STATUS5)
   END_RUNG
   // the same network as SCL:
   IF #AlwaysTrue THEN
       #STATUS1 := 'GAS BLANKETING STARTED';
       #STATUS2 := 'GAS BLANKETING PAUSED';
       #STATUS3 := 'GAS BLANKETING RESUMED';
       #STATUS4 := 'GAS BLANKETING OVER';
       #STATUS5 := 'GAS BLANKETING RESETED';
   END_IF;
END_REGION

REGION Network 9: Print Logic
   RUNG wire#powerrail
      Contact( #AlwaysTrue )
      wire#w1
      P_Contact(operand := #Selected, bit := #RE3)
      { S7_GenerateENO := "TRUE" } Move(in := 1, out1 => #PrintWord)   // 'STARTED'
      S_Move(in := #STATUS1, out => #PrintStatus)
      S_Coil( #PrintTriggerTemp )
   END_RUNG
   RUNG wire#w1
      Contact( #Selected )
      N_Contact(operand := #Running, bit := #RE4)
      I_Contact( #Reset )
      { S7_GenerateENO := "TRUE" } Move(in := 2, out1 => #PrintWord)   // 'PAUSED'
      S_Move(in := #STATUS2, out => #PrintStatus)
      wire#w2
      S_Coil( #PrintTriggerTemp )
   END_RUNG
   RUNG wire#w2
      S_Coil( #Paused )
   END_RUNG
   RUNG wire#w1
      Contact( #Selected )
      Contact( #Paused )
      P_Contact(operand := #Running, bit := #RE5)
      { S7_GenerateENO := "TRUE" } Move(in := 3, out1 => #PrintWord)   // 'RESUMED'
      S_Move(in := #STATUS3, out => #PrintStatus)
      wire#w3
      S_Coil( #PrintTriggerTemp )
   END_RUNG
   RUNG wire#w3
      R_Coil( #Paused )
   END_RUNG
   RUNG wire#w1
      P_Contact(operand := #BlanketingOver, bit := #RE6)
      { S7_GenerateENO := "TRUE" } Move(in := 4, out1 => #PrintWord)   // 'OVER'
      S_Move(in := #STATUS4, out => #PrintStatus)
      S_Coil( #PrintTriggerTemp )
   END_RUNG
   RUNG wire#w1
      P_Contact(operand := #Reset, bit := #RE7)
      { S7_GenerateENO := "TRUE" } Move(in := 5, out1 => #PrintWord)   // 'RESETED'
      S_Move(in := #STATUS5, out => #PrintStatus)
      S_Coil( #PrintTriggerTemp )
   END_RUNG
   RUNG wire#w1
      I_Contact( #Selected )
      R_Coil( #Paused )
   END_RUNG
   RUNG wire#w1
      Contact( #PrintTriggerTemp )
      Coil( #PrintTrigger )
   END_RUNG
   // the same network as SCL:
   // ENO of a box is taken as its EN; it also drops when the box reports an error
   #_w1 := #AlwaysTrue AND #Selected AND NOT #RE3;   // rising edge of #Selected
   #RE3 := #Selected;
   IF #_w1 THEN
       #PrintWord := 1;   // 'STARTED'
       #PrintStatus := #STATUS1;
       #PrintTriggerTemp := TRUE;
   END_IF;
   #_w2 := #AlwaysTrue AND #Selected AND NOT #Running AND #RE4;   // falling edge of #Running
   #RE4 := #Running;
   IF #_w2 AND NOT #Reset THEN
       #PrintWord := 2;   // 'PAUSED'
       #PrintStatus := #STATUS2;
       #PrintTriggerTemp := TRUE;
       #Paused := TRUE;
   END_IF;
   #_w3 := #AlwaysTrue AND #Selected AND #Paused AND #Running AND NOT #RE5;   // rising edge of #Running
   #RE5 := #Running;
   IF #_w3 THEN
       #PrintWord := 3;   // 'RESUMED'
       #PrintStatus := #STATUS3;
       #PrintTriggerTemp := TRUE;
       #Paused := FALSE;
   END_IF;
   #_w4 := #AlwaysTrue AND #BlanketingOver AND NOT #RE6;   // rising edge of #BlanketingOver
   #RE6 := #BlanketingOver;
   IF #_w4 THEN
       #PrintWord := 4;   // 'OVER'
       #PrintStatus := #STATUS4;
       #PrintTriggerTemp := TRUE;
   END_IF;
   #_w5 := #AlwaysTrue AND #Reset AND NOT #RE7;   // rising edge of #Reset
   #RE7 := #Reset;
   IF #_w5 THEN
       #PrintWord := 5;   // 'RESETED'
       #PrintStatus := #STATUS5;
       #PrintTriggerTemp := TRUE;
   END_IF;
   IF #AlwaysTrue AND NOT #Selected THEN #Paused := FALSE; END_IF;
   #PrintTrigger := #AlwaysTrue AND #PrintTriggerTemp;
END_REGION

REGION Network 10: Print Trigger Reset
   RUNG wire#powerrail
      Contact( #PrintTriggerTemp )
      { S7_Templates := "time_type := Time" } #PrintTriggerResetTimer.TON(pt := T#1s, et =>)
      R_Coil( #PrintTriggerTemp )
   END_RUNG
   // the same network as SCL:
   #PrintTriggerResetTimer(IN := #PrintTriggerTemp, PT := T#1s);   // TON
   IF #PrintTriggerResetTimer.Q THEN #PrintTriggerTemp := FALSE; END_IF;
END_REGION

REGION Network 11: Button Reset
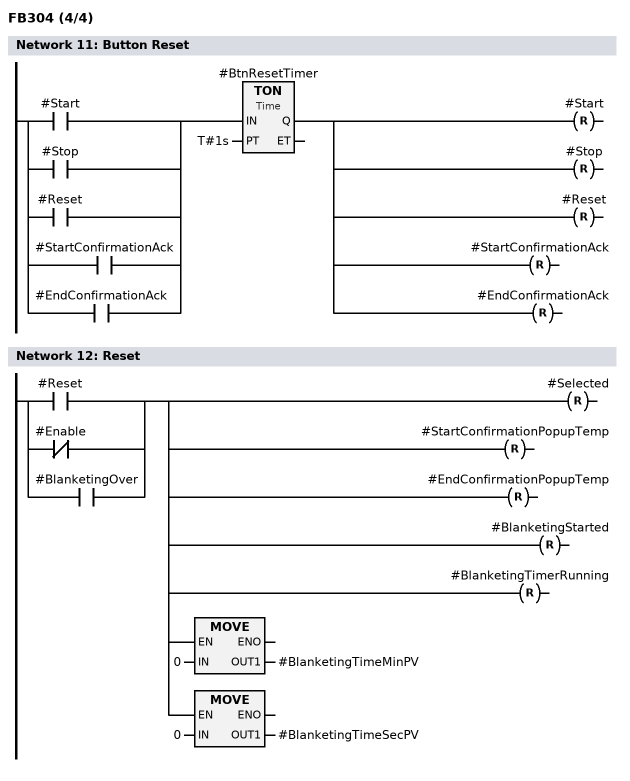
   RUNG wire#powerrail
      Contact( #Start )
      wire#w1
      { S7_Templates := "time_type := Time" } #BtnResetTimer.TON(pt := T#1s, et =>)
      wire#w2
      R_Coil( #Start )
   END_RUNG
   RUNG wire#powerrail
      Contact( #Stop )
   END_RUNG wire#w1
   RUNG wire#powerrail
      Contact( #Reset )
   END_RUNG wire#w1
   RUNG wire#powerrail
      Contact( #StartConfirmationAck )
   END_RUNG wire#w1
   RUNG wire#powerrail
      Contact( #EndConfirmationAck )
   END_RUNG wire#w1
   RUNG wire#w2
      R_Coil( #Stop )
   END_RUNG
   RUNG wire#w2
      R_Coil( #Reset )
   END_RUNG
   RUNG wire#w2
      R_Coil( #StartConfirmationAck )
   END_RUNG
   RUNG wire#w2
      R_Coil( #EndConfirmationAck )
   END_RUNG
   // the same network as SCL:
   #BtnResetTimer(IN := #Start OR #Stop OR #Reset OR #StartConfirmationAck OR #EndConfirmationAck, PT := T#1s);   // TON
   IF #BtnResetTimer.Q THEN
       #Start := FALSE;
       #Stop := FALSE;
       #Reset := FALSE;
       #StartConfirmationAck := FALSE;
       #EndConfirmationAck := FALSE;
   END_IF;
END_REGION

REGION Network 12: Reset
   RUNG wire#powerrail
      Contact( #Reset )
      wire#w1
      R_Coil( #Selected )
   END_RUNG
   RUNG wire#powerrail
      I_Contact( #Enable )
   END_RUNG wire#w1
   RUNG wire#powerrail
      Contact( #BlanketingOver )
   END_RUNG wire#w1
   RUNG wire#w1
      R_Coil( #StartConfirmationPopupTemp )
   END_RUNG
   RUNG wire#w1
      R_Coil( #EndConfirmationPopupTemp )
   END_RUNG
   RUNG wire#w1
      R_Coil( #BlanketingStarted )
   END_RUNG
   RUNG wire#w1
      R_Coil( #BlanketingTimerRunning )
   END_RUNG
   RUNG wire#w1
      { S7_GenerateENO := "TRUE" } Move(in := 0, out1 => #BlanketingTimeMinPV)
   END_RUNG
   RUNG wire#w1
      { S7_GenerateENO := "TRUE" } Move(in := 0, out1 => #BlanketingTimeSecPV)
   END_RUNG
   // the same network as SCL:
   IF #Reset OR NOT #Enable OR #BlanketingOver THEN
       #Selected := FALSE;
       #StartConfirmationPopupTemp := FALSE;
       #EndConfirmationPopupTemp := FALSE;
       #BlanketingStarted := FALSE;
       #BlanketingTimerRunning := FALSE;
       #BlanketingTimeMinPV := 0;
       #BlanketingTimeSecPV := 0;
   END_IF;
END_REGION
END_FUNCTION_BLOCK

FUNCTION_BLOCK "FB305"   // FB305, LAD
{ S7_Optimized_Access := 'TRUE' }
// stored: AutoNumber false, MemoryReserve 100, SetENOAutomatically false
   VAR_INPUT
      Enable : Bool;
      Disable : Bool;
      Fault : Bool;
      SecPulse : Bool;
      AlwaysTrue : Bool;
      StartConfirmationPopupSel : Bool;   // StartConfirmationPopupSel: 0-NO/1-YES
      EndConfirmationPopupSel : Bool;   // EndConfirmationPopupSel: 0-NO/1-YES
      WeightBasedSel : Bool;   // Weight Based Sel: 0-NO/1-YES
      AdditionMethodSel : Bool;   // Addition Method : 0-Add In Weight/1-Loss In Weight
      TransferTypeSel : Bool;   // Transfer Type Selection: 0-Complete/1-Partial
      TransferVesselPressureCheckSel : Bool;   // Transfer Vessel Pressure Check Selection: 0-NO/1-YES
      PressureReleaseSel : Bool;   // Pressure Release Selection: 0-NO/1-YES
      DelaytoEmptyLineSel : Bool;   // Delay to Empty Line Selection: 0-NO/1-YES
      FlowSwitchCheckSel : Bool;   // Flow Switch Check Selection: 0-NO/1-YES
      TransfertoFMSel : Bool;   // Transfer to FM Selection: 0-NO/1-YES
      RecBasedTransferSel : Bool;   // Recirculation Based Transfer Selection: 0-NO/1-YES
      TemperatureControlSel : Bool;   // Temperature Control Selection: 0-NO/1-YES
      TransferMethodSel : Int;   // 0-Pump/ 1-Pressure/2-Vacuum/3-Pump+Pressure/4-Pump+Vacuum/5-Pressure+Vacuum
      GasSel : Int;   // Gas Selection - 0-AIR/1-N2
      SetPressure : Real := 1.0;
      SetVacuum : Real := -300.0;
      SetQuantity : Real := 10.0;   // Weight Based Sel: 1-YES
      SetSpeed : Real := 100.0;
      ActualPressure : Real;
      ActualVacuum : Real;
      ActualQuantity : Real;   // Collecting Vessel Weight
      ActualQuantityVessel : Real;   // Transffering Vessel Weight
      FlowSwitchInput : Bool;
      FMHealthyInput : Bool;
      TemperatureReachedInput : Bool;
      PressureTol : Real := 0.3;
      VacuumTol : Real := 10.0;
      InflightQuantity : Real;
      VesselEmptyWeight : Real;
      DelaytoEmptyLine : Int := 10;
      DelaytoReleaseTransferVesselPressure : Int := 10;
      DelaytoReleasePressure : Int := 10;
      DelaytoStartPump : Int := 0;
      DelaytoOpenGasIn : Int := 3;
   END_VAR
   VAR_OUTPUT
      AirValve : Bool;
      N2Valve : Bool;
      VacuumInValve : Bool;
      VacuumLineValves : Bool;
      LineValves : Bool;
      SuctionInValve : Bool;
      VesselOutletValve : Bool;
      RecirculationLineValves : Bool;
      FMInValve : Bool;
      PumpCmd : Bool;
      VacuumPumpCmd : Bool;
      StartConfirmationPopup : Bool;   // For Start Confirmation Popup Selection: Yes
      EndConfirmationPopup : Bool;   // For End Confirmation Popup Selection: Yes
      ActualSpeed : Real;
      PrintTrigger : Bool;
      PrintWord : Int;
      PrintStatus : String[50];
   END_VAR
   VAR_IN_OUT
      Start : Bool;
      Stop : Bool;
      Reset : Bool;
      StartConfirmationAck : Bool;   // For Start Confirmation Popup Selection: Yes
      EndConfirmationAck : Bool;   // For End Confirmation Popup Selection: Yes
      SpareBtn1 : Bool;
      SpareBtn2 : Bool;
      SpareBtn3 : Bool;
      Running : Bool;
      Selected : Bool;
      Paused : Bool;
      StartConfirmationPopupTemp : Bool;   // For Start Confirmation Popup Selection: Yes
      EndConfirmationPopupTemp : Bool;   // For End Confirmation Popup Selection: Yes
      Started : Bool;
      Over : Bool;
      PumpBasedSelected : Bool;
      PressureBasedSelected : Bool;
      VacuumBasedSelected : Bool;
      StartDelaytoEmptyLine : Bool;
      StartDelaytoReleasePressure : Bool;
      SecondPopup : Bool;
      SecondPopupAck : Bool;
      PressureTolNeg : Real;   // VacuumTolNeg - For unit "mmHg" / PressureTolNeg - For unit "bar"
      VacuumTolNeg : Real;   // VacuumTolNeg - For unit "mmHg" / PressureTolNeg - For unit "bar"
      ActualSetQuantityCalc : Real;   // For WeightBaseSel: 1-YES
      ActualSetQuantity : Real;   // For WeightBaseSel: 1-YES
   END_VAR
   VAR
      ValveOnDelayPV : Int;
      ValveOffDelayPV : Int;
      PrintTriggerTemp : Bool;
      RE1 : Bool;
      RE2 : Bool;
      RE3 : Bool;
      RE4 : Bool;
      RE5 : Bool;
      RE6 : Bool;
      RE7 : Bool;
      PrintTriggerResetTimer { S7_SetPoint := 'True'} : TON_TIME;
      BtnResetTimer { S7_SetPoint := 'True'} : TON_TIME;
      TransferVesselPressureCheckDelay { S7_SetPoint := 'True'} : "FB103";
      PressureReleaseDelay { S7_SetPoint := 'True'} : "FB103";
      EmptyLineDelay { S7_SetPoint := 'True'} : "FB103";
      PumpOnDelayPv { S7_SetPoint := 'True'} : Int;
   END_VAR
   VAR_TEMP
      STATUS1 : String[40];
      STATUS2 : String[40];
      STATUS3 : String[40];
      STATUS4 : String[40];
      STATUS5 : String[40];
      STATUS6 : String[40];
   END_VAR
   VAR CONSTANT
      PumpOnDelay : Int;
      PumpOffDelay : Int;
   END_VAR
   VAR_TEMP   // added for the SCL form of the ladder/FBD networks
      _w1 : Bool;
      _w2 : Bool;
      _w3 : Bool;
      _w4 : Bool;
      _w5 : Bool;
      _w6 : Bool;
   END_VAR
BEGIN

REGION Network 2: Running
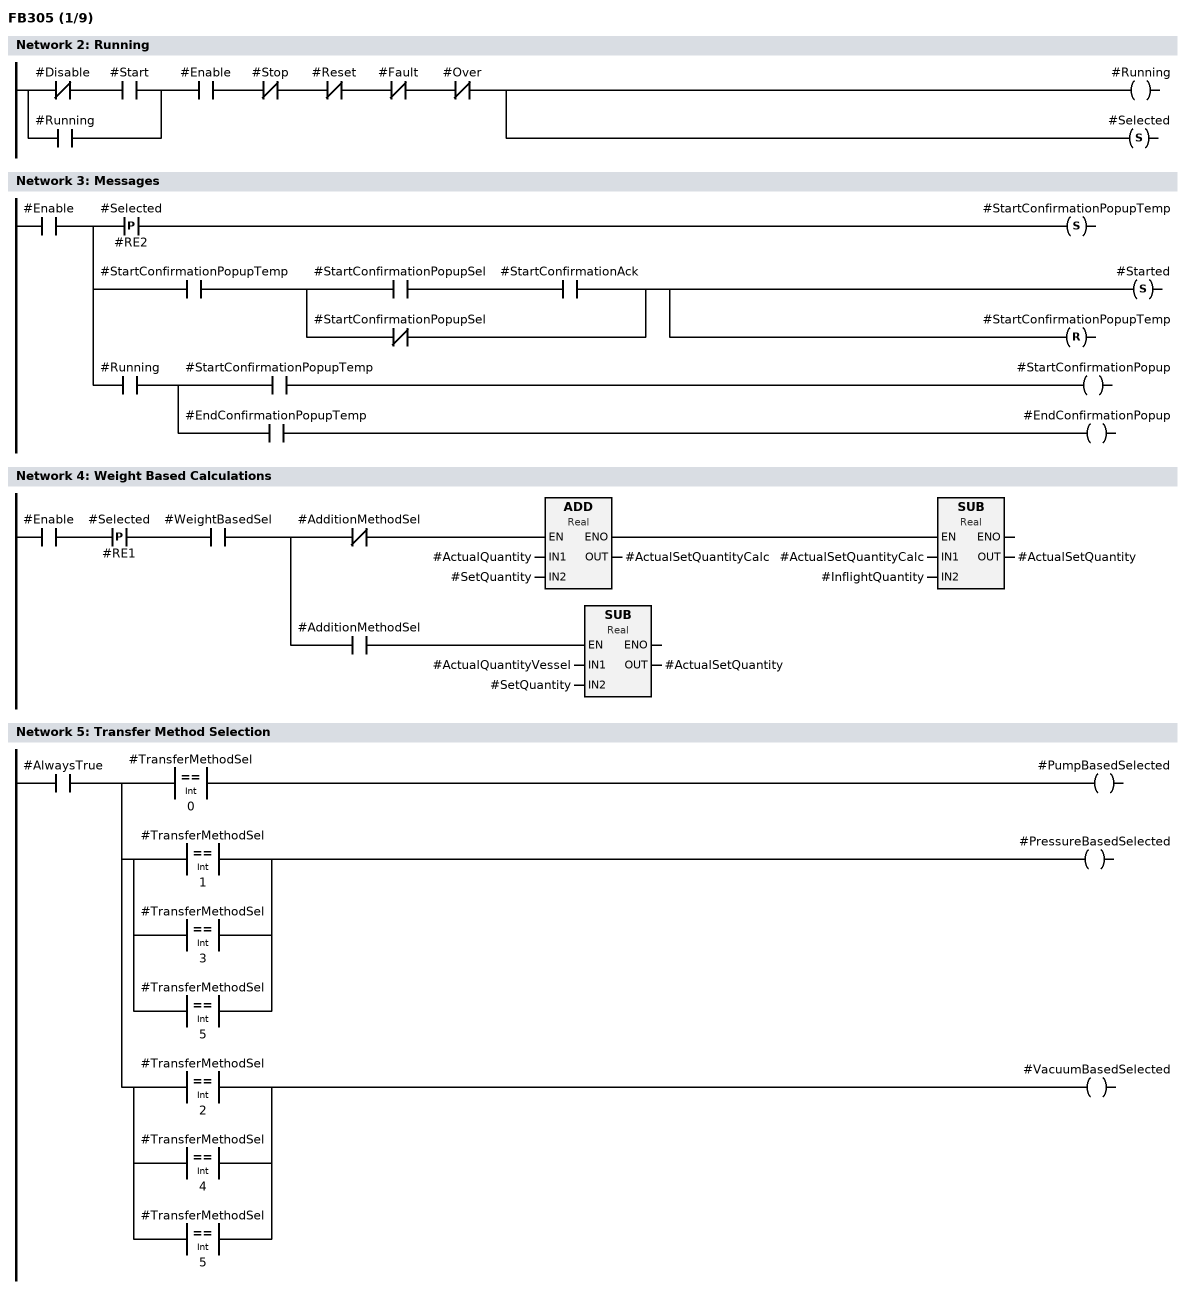
   RUNG wire#powerrail
      I_Contact( #Disable )
      Contact( #Start )
      wire#w1
      Contact( #Enable )
      I_Contact( #Stop )
      I_Contact( #Reset )
      I_Contact( #Fault )
      I_Contact( #Over )
      wire#w2
      Coil( #Running )
   END_RUNG
   RUNG wire#powerrail
      Contact( #Running )
   END_RUNG wire#w1
   RUNG wire#w2
      S_Coil( #Selected )
   END_RUNG
   // the same network as SCL:
   #Running := ((NOT #Disable AND #Start) OR #Running) AND #Enable AND NOT #Stop AND NOT #Reset AND NOT #Fault AND NOT #Over;
   IF #Running THEN #Selected := TRUE; END_IF;
END_REGION

REGION Network 3: Messages
   RUNG wire#powerrail
      Contact( #Enable )
      wire#w1
      P_Contact(operand := #Selected, bit := #RE2)
      S_Coil( #StartConfirmationPopupTemp )
   END_RUNG
   RUNG wire#w1
      Contact( #StartConfirmationPopupTemp )
      wire#w2
      Contact( #StartConfirmationPopupSel )
      Contact( #StartConfirmationAck )
      wire#w3
      S_Coil( #Started )
   END_RUNG
   RUNG wire#w2
      I_Contact( #StartConfirmationPopupSel )
   END_RUNG wire#w3
   RUNG wire#w3
      R_Coil( #StartConfirmationPopupTemp )
   END_RUNG
   RUNG wire#w1
      Contact( #Running )
      wire#w4
      Contact( #StartConfirmationPopupTemp )
      Coil( #StartConfirmationPopup )
   END_RUNG
   RUNG wire#w4
      Contact( #EndConfirmationPopupTemp )
      Coil( #EndConfirmationPopup )
   END_RUNG
   // the same network as SCL:
   #_w1 := #Enable AND #Selected AND NOT #RE2;   // rising edge of #Selected
   #RE2 := #Selected;
   IF #_w1 THEN #StartConfirmationPopupTemp := TRUE; END_IF;
   IF #Enable AND #StartConfirmationPopupTemp AND ((#StartConfirmationPopupSel AND #StartConfirmationAck) OR NOT #StartConfirmationPopupSel) THEN
       #Started := TRUE;
       #StartConfirmationPopupTemp := FALSE;
   END_IF;
   #_w2 := #Enable AND #Running;
   #StartConfirmationPopup := #_w2 AND #StartConfirmationPopupTemp;
   #EndConfirmationPopup := #_w2 AND #EndConfirmationPopupTemp;
END_REGION

REGION Network 4: Weight Based Calculations
   RUNG wire#powerrail
      Contact( #Enable )
      P_Contact(operand := #Selected, bit := #RE1)
      Contact( #WeightBasedSel )
      wire#w1
      I_Contact( #AdditionMethodSel )
      { S7_Templates := "SrcType := Real"; S7_GenerateENO := "TRUE" } Add(in1 := #ActualQuantity, in2 := #SetQuantity, out => #ActualSetQuantityCalc)
      { S7_Templates := "SrcType := Real"; S7_GenerateENO := "TRUE" } Sub(in1 := #ActualSetQuantityCalc, in2 := #InflightQuantity, out => #ActualSetQuantity)
   END_RUNG
   RUNG wire#w1
      Contact( #AdditionMethodSel )
      { S7_Templates := "SrcType := Real"; S7_GenerateENO := "TRUE" } Sub(in1 := #ActualQuantityVessel, in2 := #SetQuantity, out => #ActualSetQuantity)
   END_RUNG
   // the same network as SCL:
   // ENO of a box is taken as its EN; it also drops when the box reports an error
   #_w1 := #Enable AND #Selected AND NOT #RE1;   // rising edge of #Selected
   #RE1 := #Selected;
   #_w2 := #_w1 AND #WeightBasedSel;
   IF #_w2 AND NOT #AdditionMethodSel THEN
       #ActualSetQuantityCalc := #ActualQuantity + #SetQuantity;
       #ActualSetQuantity := #ActualSetQuantityCalc - #InflightQuantity;
   END_IF;
   IF #_w2 AND #AdditionMethodSel THEN #ActualSetQuantity := #ActualQuantityVessel - #SetQuantity; END_IF;
END_REGION

REGION Network 5: Transfer Method Selection
   RUNG wire#powerrail
      Contact( #AlwaysTrue )
      wire#w1
      { S7_Templates := "SrcType := Int" } EQ_Contact(in1 := #TransferMethodSel, in2 := 0)
      Coil( #PumpBasedSelected )
   END_RUNG
   RUNG wire#w1
      { S7_Templates := "SrcType := Int" } EQ_Contact(in1 := #TransferMethodSel, in2 := 1)
      wire#w2
      Coil( #PressureBasedSelected )
   END_RUNG
   RUNG wire#w1
      { S7_Templates := "SrcType := Int" } EQ_Contact(in1 := #TransferMethodSel, in2 := 3)
   END_RUNG wire#w2
   RUNG wire#w1
      { S7_Templates := "SrcType := Int" } EQ_Contact(in1 := #TransferMethodSel, in2 := 5)
   END_RUNG wire#w2
   RUNG wire#w1
      { S7_Templates := "SrcType := Int" } EQ_Contact(in1 := #TransferMethodSel, in2 := 2)
      wire#w3
      Coil( #VacuumBasedSelected )
   END_RUNG
   RUNG wire#w1
      { S7_Templates := "SrcType := Int" } EQ_Contact(in1 := #TransferMethodSel, in2 := 4)
   END_RUNG wire#w3
   RUNG wire#w1
      { S7_Templates := "SrcType := Int" } EQ_Contact(in1 := #TransferMethodSel, in2 := 5)
   END_RUNG wire#w3
   // the same network as SCL:
   #PumpBasedSelected := #AlwaysTrue AND (#TransferMethodSel = 0);
   #PressureBasedSelected := #AlwaysTrue AND ((#TransferMethodSel = 1) OR (#TransferMethodSel = 3) OR (#TransferMethodSel = 5));
   #VacuumBasedSelected := #AlwaysTrue AND ((#TransferMethodSel = 2) OR (#TransferMethodSel = 4) OR (#TransferMethodSel = 5));
END_REGION

REGION Network 6: Negative Tolerance
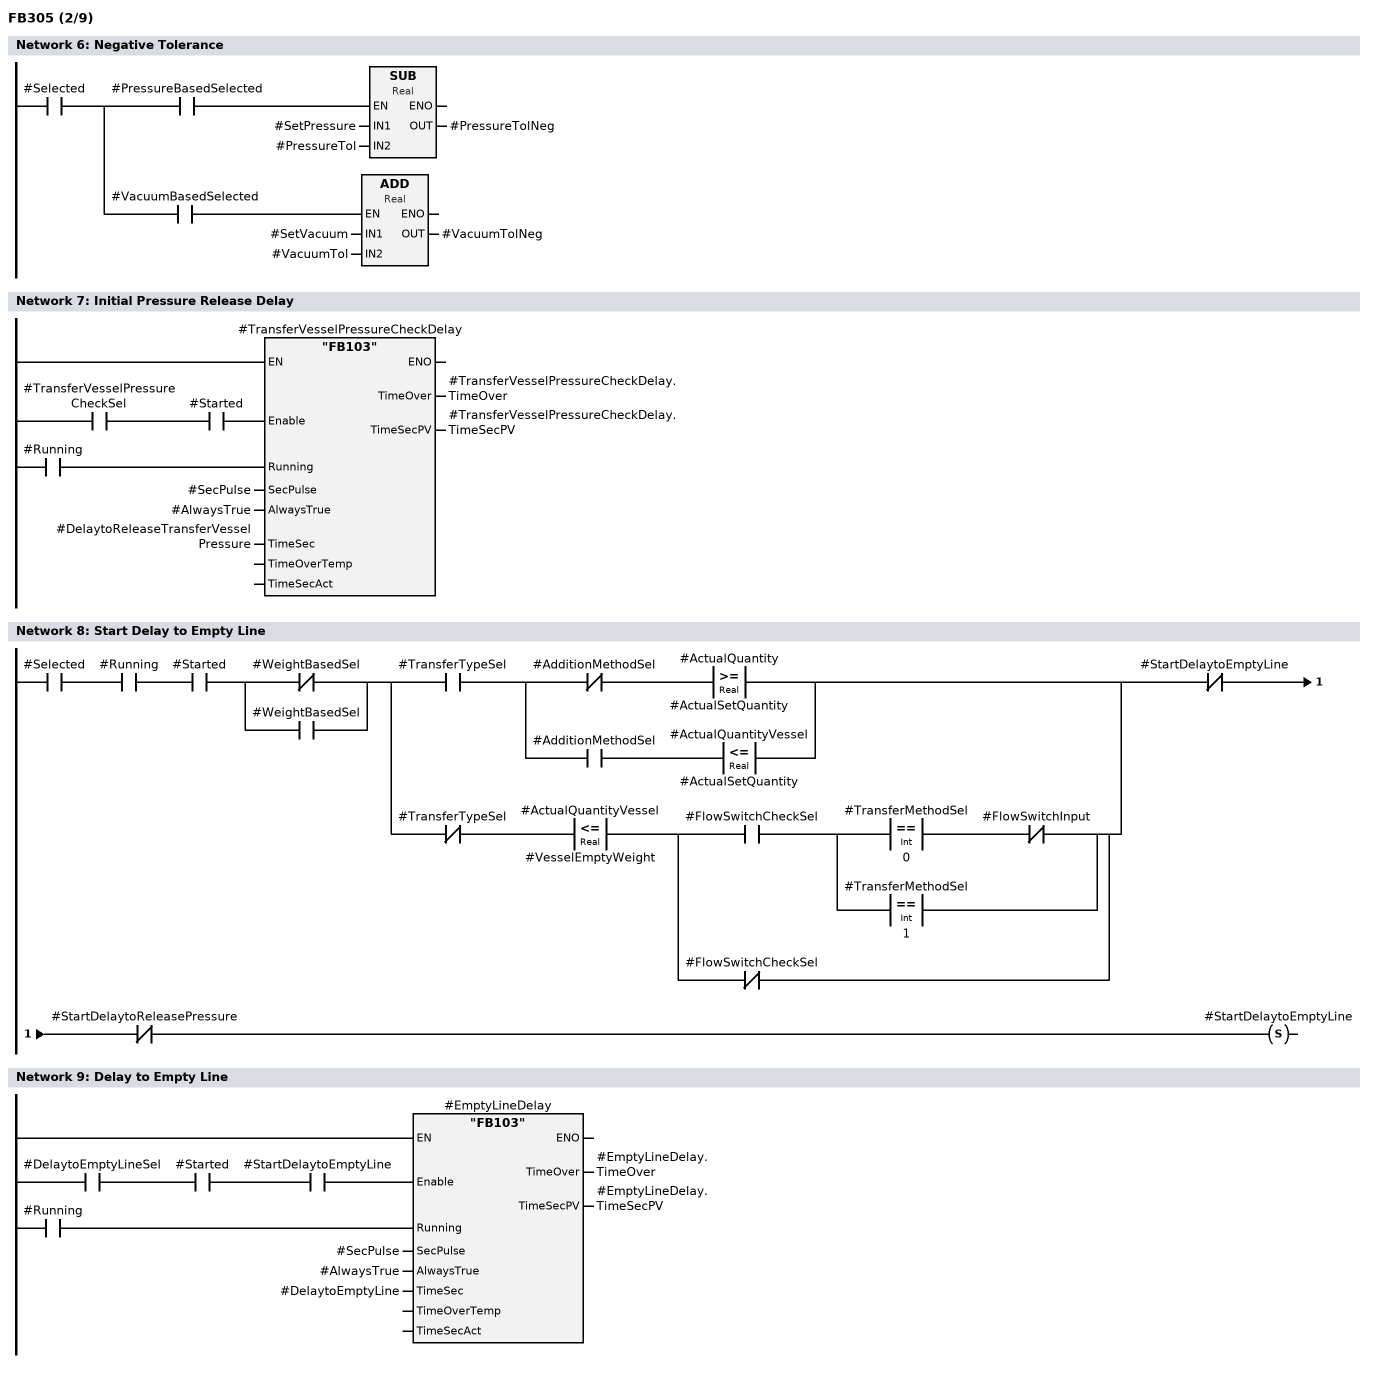
   RUNG wire#powerrail
      Contact( #Selected )
      wire#w1
      Contact( #PressureBasedSelected )
      { S7_Templates := "SrcType := Real"; S7_GenerateENO := "TRUE" } Sub(in1 := #SetPressure, in2 := #PressureTol, out => #PressureTolNeg)
   END_RUNG
   RUNG wire#w1
      Contact( #VacuumBasedSelected )
      { S7_Templates := "SrcType := Real"; S7_GenerateENO := "TRUE" } Add(in1 := #SetVacuum, in2 := #VacuumTol, out => #VacuumTolNeg)
   END_RUNG
   // the same network as SCL:
   IF #Selected AND #PressureBasedSelected THEN #PressureTolNeg := #SetPressure - #PressureTol; END_IF;
   IF #Selected AND #VacuumBasedSelected THEN #VacuumTolNeg := #SetVacuum + #VacuumTol; END_IF;
END_REGION

REGION Network 7: Initial Pressure Release Delay
   RUNG wire#powerrail
      #TransferVesselPressureCheckDelay(Enable := wire#w1, Running := wire#w2, SecPulse := #SecPulse, AlwaysTrue := #AlwaysTrue, TimeSec := #DelaytoReleaseTransferVesselPressure, TimeOverTemp :=, TimeSecAct :=, TimeOver => #TransferVesselPressureCheckDelay.TimeOver, TimeSecPV => #TransferVesselPressureCheckDelay.TimeSecPV)
   END_RUNG
   RUNG wire#powerrail
      Contact( #TransferVesselPressureCheckSel )
      Contact( #Started )
   END_RUNG wire#w1
   RUNG wire#powerrail
      Contact( #Running )
   END_RUNG wire#w2
   // the same network as SCL:
   #TransferVesselPressureCheckDelay(Enable := #TransferVesselPressureCheckSel AND #Started,   // "FB103"
                           Running := #Running,
                           SecPulse := #SecPulse,
                           AlwaysTrue := #AlwaysTrue,
                           TimeSec := #DelaytoReleaseTransferVesselPressure,
                           TimeOver => #TransferVesselPressureCheckDelay.TimeOver,
                           TimeSecPV => #TransferVesselPressureCheckDelay.TimeSecPV);
END_REGION

REGION Network 8: Start Delay to Empty Line
   RUNG wire#powerrail
      Contact( #Selected )
      Contact( #Running )
      Contact( #Started )
      wire#w1
      I_Contact( #WeightBasedSel )
      wire#w2
      Contact( #TransferTypeSel )
      wire#w3
      I_Contact( #AdditionMethodSel )
      { S7_Templates := "SrcType := Real" } GE_Contact(in1 := #ActualQuantity, in2 := #ActualSetQuantity)
      wire#w4
      I_Contact( #StartDelaytoEmptyLine )
      I_Contact( #StartDelaytoReleasePressure )
      S_Coil( #StartDelaytoEmptyLine )
   END_RUNG
   RUNG wire#w1
      Contact( #WeightBasedSel )
   END_RUNG wire#w2
   RUNG wire#w3
      Contact( #AdditionMethodSel )
      { S7_Templates := "SrcType := Real" } LE_Contact(in1 := #ActualQuantityVessel, in2 := #ActualSetQuantity)
   END_RUNG wire#w4
   RUNG wire#w2
      I_Contact( #TransferTypeSel )
      { S7_Templates := "SrcType := Real" } LE_Contact(in1 := #ActualQuantityVessel, in2 := #VesselEmptyWeight)
      wire#w5
      Contact( #FlowSwitchCheckSel )
      wire#w6
      { S7_Templates := "SrcType := Int" } EQ_Contact(in1 := #TransferMethodSel, in2 := 0)
      I_Contact( #FlowSwitchInput )
   END_RUNG wire#w4
   RUNG wire#w6
      { S7_Templates := "SrcType := Int" } EQ_Contact(in1 := #TransferMethodSel, in2 := 1)
   END_RUNG wire#w4
   RUNG wire#w5
      I_Contact( #FlowSwitchCheckSel )
   END_RUNG wire#w4
   // the same network as SCL:
   IF #Selected AND #Running AND #Started AND (NOT #WeightBasedSel OR #WeightBasedSel) AND ((#TransferTypeSel AND ((NOT #AdditionMethodSel AND (#ActualQuantity >= #ActualSetQuantity)) OR (#AdditionMethodSel AND (#ActualQuantityVessel <= #ActualSetQuantity)))) OR (NOT #TransferTypeSel AND (#ActualQuantityVessel <= #VesselEmptyWeight) AND ((#FlowSwitchCheckSel AND (((#TransferMethodSel = 0) AND NOT #FlowSwitchInput) OR (#TransferMethodSel = 1))) OR NOT #FlowSwitchCheckSel))) AND NOT #StartDelaytoEmptyLine AND NOT #StartDelaytoReleasePressure THEN
       #StartDelaytoEmptyLine := TRUE;
   END_IF;
END_REGION

REGION Network 9: Delay to Empty Line
   RUNG wire#powerrail
      #EmptyLineDelay(Enable := wire#w1, Running := wire#w2, SecPulse := #SecPulse, AlwaysTrue := #AlwaysTrue, TimeSec := #DelaytoEmptyLine, TimeOverTemp :=, TimeSecAct :=, TimeOver => #EmptyLineDelay.TimeOver, TimeSecPV => #EmptyLineDelay.TimeSecPV)
   END_RUNG
   RUNG wire#powerrail
      Contact( #DelaytoEmptyLineSel )
      Contact( #Started )
      Contact( #StartDelaytoEmptyLine )
   END_RUNG wire#w1
   RUNG wire#powerrail
      Contact( #Running )
   END_RUNG wire#w2
   // the same network as SCL:
   #EmptyLineDelay(Enable := #DelaytoEmptyLineSel AND #Started AND #StartDelaytoEmptyLine,   // "FB103"
                   Running := #Running,
                   SecPulse := #SecPulse,
                   AlwaysTrue := #AlwaysTrue,
                   TimeSec := #DelaytoEmptyLine,
                   TimeOver => #EmptyLineDelay.TimeOver,
                   TimeSecPV => #EmptyLineDelay.TimeSecPV);
END_REGION

REGION Network 10: Start Delay to Release After Pressure
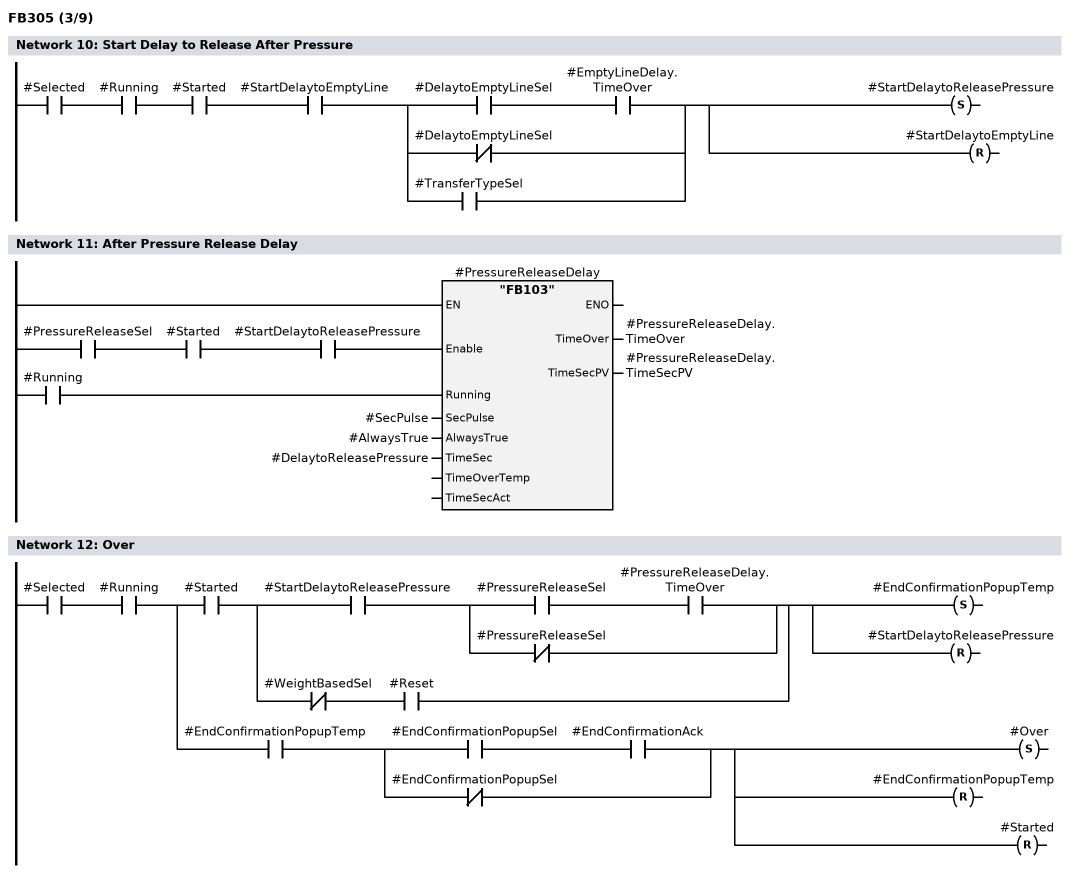
   RUNG wire#powerrail
      Contact( #Selected )
      Contact( #Running )
      Contact( #Started )
      Contact( #StartDelaytoEmptyLine )
      wire#w1
      Contact( #DelaytoEmptyLineSel )
      Contact( #EmptyLineDelay.TimeOver )
      wire#w2
      S_Coil( #StartDelaytoReleasePressure )
   END_RUNG
   RUNG wire#w1
      I_Contact( #DelaytoEmptyLineSel )
   END_RUNG wire#w2
   RUNG wire#w1
      Contact( #TransferTypeSel )
   END_RUNG wire#w2
   RUNG wire#w2
      R_Coil( #StartDelaytoEmptyLine )
   END_RUNG
   // the same network as SCL:
   IF #Selected AND #Running AND #Started AND #StartDelaytoEmptyLine AND ((#DelaytoEmptyLineSel AND #EmptyLineDelay.TimeOver) OR NOT #DelaytoEmptyLineSel OR #TransferTypeSel) THEN
       #StartDelaytoReleasePressure := TRUE;
       #StartDelaytoEmptyLine := FALSE;
   END_IF;
END_REGION

REGION Network 11: After Pressure Release Delay
   RUNG wire#powerrail
      #PressureReleaseDelay(Enable := wire#w1, Running := wire#w2, SecPulse := #SecPulse, AlwaysTrue := #AlwaysTrue, TimeSec := #DelaytoReleasePressure, TimeOverTemp :=, TimeSecAct :=, TimeOver => #PressureReleaseDelay.TimeOver, TimeSecPV => #PressureReleaseDelay.TimeSecPV)
   END_RUNG
   RUNG wire#powerrail
      Contact( #PressureReleaseSel )
      Contact( #Started )
      Contact( #StartDelaytoReleasePressure )
   END_RUNG wire#w1
   RUNG wire#powerrail
      Contact( #Running )
   END_RUNG wire#w2
   // the same network as SCL:
   #PressureReleaseDelay(Enable := #PressureReleaseSel AND #Started AND #StartDelaytoReleasePressure,   // "FB103"
                         Running := #Running,
                         SecPulse := #SecPulse,
                         AlwaysTrue := #AlwaysTrue,
                         TimeSec := #DelaytoReleasePressure,
                         TimeOver => #PressureReleaseDelay.TimeOver,
                         TimeSecPV => #PressureReleaseDelay.TimeSecPV);
END_REGION

REGION Network 12: Over
   RUNG wire#powerrail
      Contact( #Selected )
      Contact( #Running )
      wire#w1
      Contact( #Started )
      wire#w2
      Contact( #StartDelaytoReleasePressure )
      wire#w3
      Contact( #PressureReleaseSel )
      Contact( #PressureReleaseDelay.TimeOver )
      wire#w4
      S_Coil( #EndConfirmationPopupTemp )
   END_RUNG
   RUNG wire#w3
      I_Contact( #PressureReleaseSel )
   END_RUNG wire#w4
   RUNG wire#w2
      I_Contact( #WeightBasedSel )
      Contact( #Reset )
   END_RUNG wire#w4
   RUNG wire#w4
      R_Coil( #StartDelaytoReleasePressure )
   END_RUNG
   RUNG wire#w1
      Contact( #EndConfirmationPopupTemp )
      wire#w5
      Contact( #EndConfirmationPopupSel )
      Contact( #EndConfirmationAck )
      wire#w6
      S_Coil( #Over )
   END_RUNG
   RUNG wire#w5
      I_Contact( #EndConfirmationPopupSel )
   END_RUNG wire#w6
   RUNG wire#w6
      R_Coil( #EndConfirmationPopupTemp )
   END_RUNG
   RUNG wire#w6
      R_Coil( #Started )
   END_RUNG
   // the same network as SCL:
   #_w1 := #Selected AND #Running;
   IF #_w1 AND #Started AND ((#StartDelaytoReleasePressure AND ((#PressureReleaseSel AND #PressureReleaseDelay.TimeOver) OR NOT #PressureReleaseSel)) OR (NOT #WeightBasedSel AND #Reset)) THEN
       #EndConfirmationPopupTemp := TRUE;
       #StartDelaytoReleasePressure := FALSE;
   END_IF;
   IF #_w1 AND #EndConfirmationPopupTemp AND ((#EndConfirmationPopupSel AND #EndConfirmationAck) OR NOT #EndConfirmationPopupSel) THEN
       #Over := TRUE;
   END_IF;
   #_w2 := #_w1 AND #EndConfirmationPopupTemp AND ((#EndConfirmationPopupSel AND #EndConfirmationAck) OR NOT #EndConfirmationPopupSel);
   IF #_w2 THEN
       #EndConfirmationPopupTemp := FALSE;
       #Started := FALSE;
   END_IF;
END_REGION

REGION Network 13: Output On
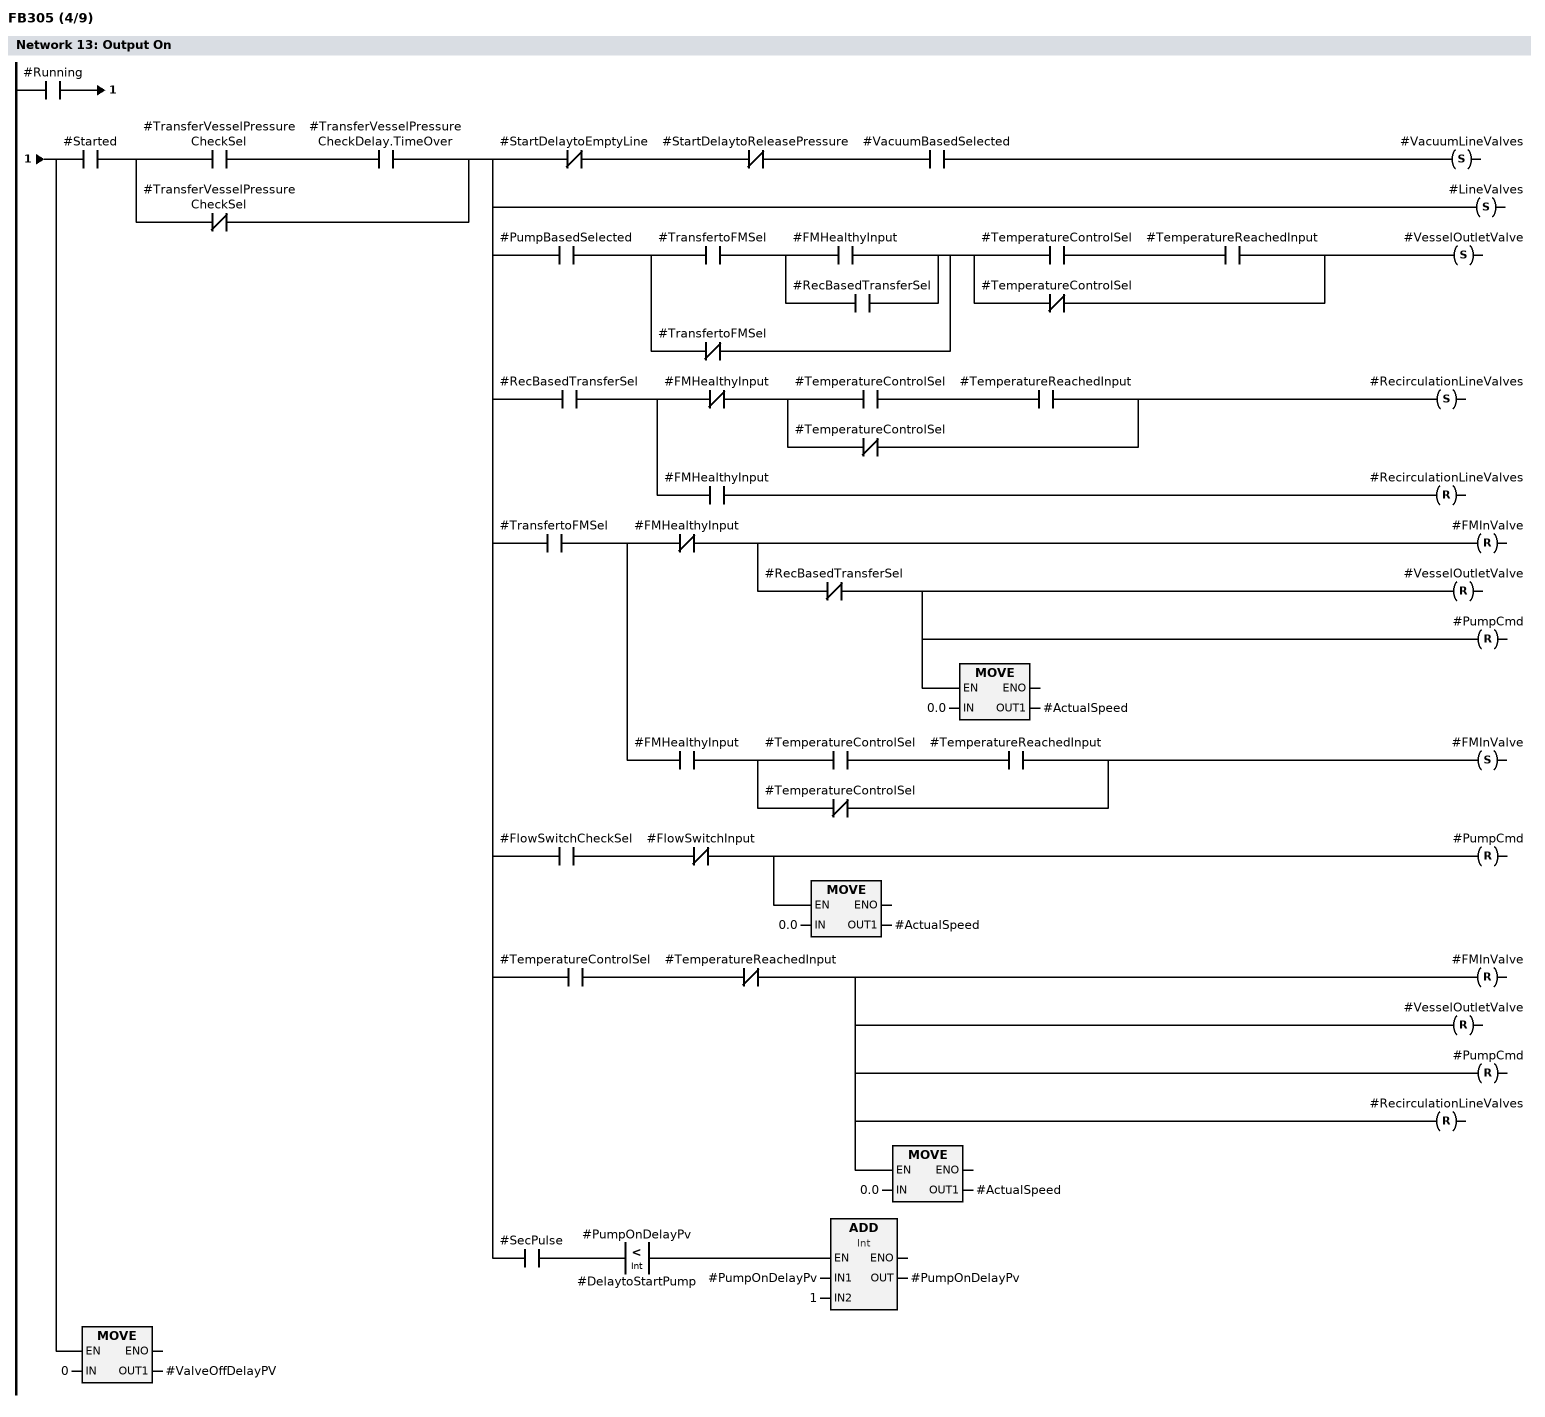
   RUNG wire#powerrail
      Contact( #Running )
      wire#w1
      Contact( #Started )
      wire#w2
      Contact( #TransferVesselPressureCheckSel )
      Contact( #TransferVesselPressureCheckDelay.TimeOver )
      wire#w3
      I_Contact( #StartDelaytoEmptyLine )
      I_Contact( #StartDelaytoReleasePressure )
      Contact( #VacuumBasedSelected )
      S_Coil( #VacuumLineValves )
   END_RUNG
   RUNG wire#w2
      I_Contact( #TransferVesselPressureCheckSel )
   END_RUNG wire#w3
   RUNG wire#w3
      S_Coil( #LineValves )
   END_RUNG
   RUNG wire#w3
      Contact( #PumpBasedSelected )
      wire#w4
      Contact( #TransfertoFMSel )
      wire#w5
      Contact( #FMHealthyInput )
      wire#w6
      Contact( #TemperatureControlSel )
      Contact( #TemperatureReachedInput )
      wire#w7
      S_Coil( #VesselOutletValve )
   END_RUNG
   RUNG wire#w5
      Contact( #RecBasedTransferSel )
   END_RUNG wire#w6
   RUNG wire#w4
      I_Contact( #TransfertoFMSel )
   END_RUNG wire#w6
   RUNG wire#w6
      I_Contact( #TemperatureControlSel )
   END_RUNG wire#w7
   RUNG wire#w3
      Contact( #RecBasedTransferSel )
      wire#w8
      I_Contact( #FMHealthyInput )
      wire#w9
      Contact( #TemperatureControlSel )
      Contact( #TemperatureReachedInput )
      wire#w10
      S_Coil( #RecirculationLineValves )
   END_RUNG
   RUNG wire#w9
      I_Contact( #TemperatureControlSel )
   END_RUNG wire#w10
   RUNG wire#w8
      Contact( #FMHealthyInput )
      R_Coil( #RecirculationLineValves )
   END_RUNG
   RUNG wire#w3
      Contact( #TransfertoFMSel )
      wire#w11
      I_Contact( #FMHealthyInput )
      wire#w12
      R_Coil( #FMInValve )
   END_RUNG
   RUNG wire#w12
      I_Contact( #RecBasedTransferSel )
      wire#w13
      R_Coil( #VesselOutletValve )
   END_RUNG
   RUNG wire#w13
      R_Coil( #PumpCmd )
   END_RUNG
   RUNG wire#w13
      Move(in := 0.0, out1 => #ActualSpeed)
   END_RUNG
   RUNG wire#w11
      Contact( #FMHealthyInput )
      wire#w14
      Contact( #TemperatureControlSel )
      Contact( #TemperatureReachedInput )
      wire#w15
      S_Coil( #FMInValve )
   END_RUNG
   RUNG wire#w14
      I_Contact( #TemperatureControlSel )
   END_RUNG wire#w15
   RUNG wire#w3
      Contact( #FlowSwitchCheckSel )
      I_Contact( #FlowSwitchInput )
      wire#w16
      R_Coil( #PumpCmd )
   END_RUNG
   RUNG wire#w16
      Move(in := 0.0, out1 => #ActualSpeed)
   END_RUNG
   RUNG wire#w3
      Contact( #TemperatureControlSel )
      I_Contact( #TemperatureReachedInput )
      wire#w17
      R_Coil( #FMInValve )
   END_RUNG
   RUNG wire#w17
      R_Coil( #VesselOutletValve )
   END_RUNG
   RUNG wire#w17
      R_Coil( #PumpCmd )
   END_RUNG
   RUNG wire#w17
      R_Coil( #RecirculationLineValves )
   END_RUNG
   RUNG wire#w17
      Move(in := 0.0, out1 => #ActualSpeed)
   END_RUNG
   RUNG wire#w3
      Contact( #SecPulse )
      { S7_Templates := "SrcType := Int" } LT_Contact(in1 := #PumpOnDelayPv, in2 := #DelaytoStartPump)
      { S7_Templates := "SrcType := Int"; S7_GenerateENO := "TRUE" } Add(in1 := #PumpOnDelayPv, in2 := 1, out => #PumpOnDelayPv)
   END_RUNG
   RUNG wire#w1
      { S7_GenerateENO := "TRUE" } Move(in := 0, out1 => #ValveOffDelayPV)
   END_RUNG
   // the same network as SCL:
   #_w1 := #Running AND #Started AND ((#TransferVesselPressureCheckSel AND #TransferVesselPressureCheckDelay.TimeOver) OR NOT #TransferVesselPressureCheckSel);
   IF #_w1 AND NOT #StartDelaytoEmptyLine AND NOT #StartDelaytoReleasePressure AND #VacuumBasedSelected THEN
       #VacuumLineValves := TRUE;
   END_IF;
   IF #_w1 THEN #LineValves := TRUE; END_IF;
   IF #_w1 AND #PumpBasedSelected AND ((#TransfertoFMSel AND (#FMHealthyInput OR #RecBasedTransferSel)) OR NOT #TransfertoFMSel) AND ((#TemperatureControlSel AND #TemperatureReachedInput) OR NOT #TemperatureControlSel) THEN
       #VesselOutletValve := TRUE;
   END_IF;
   #_w2 := #_w1 AND #RecBasedTransferSel;
   IF #_w2 AND NOT #FMHealthyInput AND ((#TemperatureControlSel AND #TemperatureReachedInput) OR NOT #TemperatureControlSel) THEN
       #RecirculationLineValves := TRUE;
   END_IF;
   IF #_w2 AND #FMHealthyInput THEN #RecirculationLineValves := FALSE; END_IF;
   #_w3 := #_w1 AND #TransfertoFMSel;
   #_w4 := #_w3 AND NOT #FMHealthyInput;
   IF #_w4 THEN #FMInValve := FALSE; END_IF;
   IF #_w4 AND NOT #RecBasedTransferSel THEN
       #VesselOutletValve := FALSE;
       #PumpCmd := FALSE;
       #ActualSpeed := 0.0;
   END_IF;
   IF #_w3 AND #FMHealthyInput AND ((#TemperatureControlSel AND #TemperatureReachedInput) OR NOT #TemperatureControlSel) THEN
       #FMInValve := TRUE;
   END_IF;
   IF #_w1 AND #FlowSwitchCheckSel AND NOT #FlowSwitchInput THEN
       #PumpCmd := FALSE;
       #ActualSpeed := 0.0;
   END_IF;
   IF #_w1 AND #TemperatureControlSel AND NOT #TemperatureReachedInput THEN
       #FMInValve := FALSE;
       #VesselOutletValve := FALSE;
       #PumpCmd := FALSE;
       #RecirculationLineValves := FALSE;
       #ActualSpeed := 0.0;
   END_IF;
   IF #_w1 AND #SecPulse AND (#PumpOnDelayPv < #DelaytoStartPump) THEN
       #PumpOnDelayPv := #PumpOnDelayPv + 1;
   END_IF;
   IF #Running THEN #ValveOffDelayPV := 0; END_IF;
END_REGION

REGION Network 14: Output On When Pump Based Selection
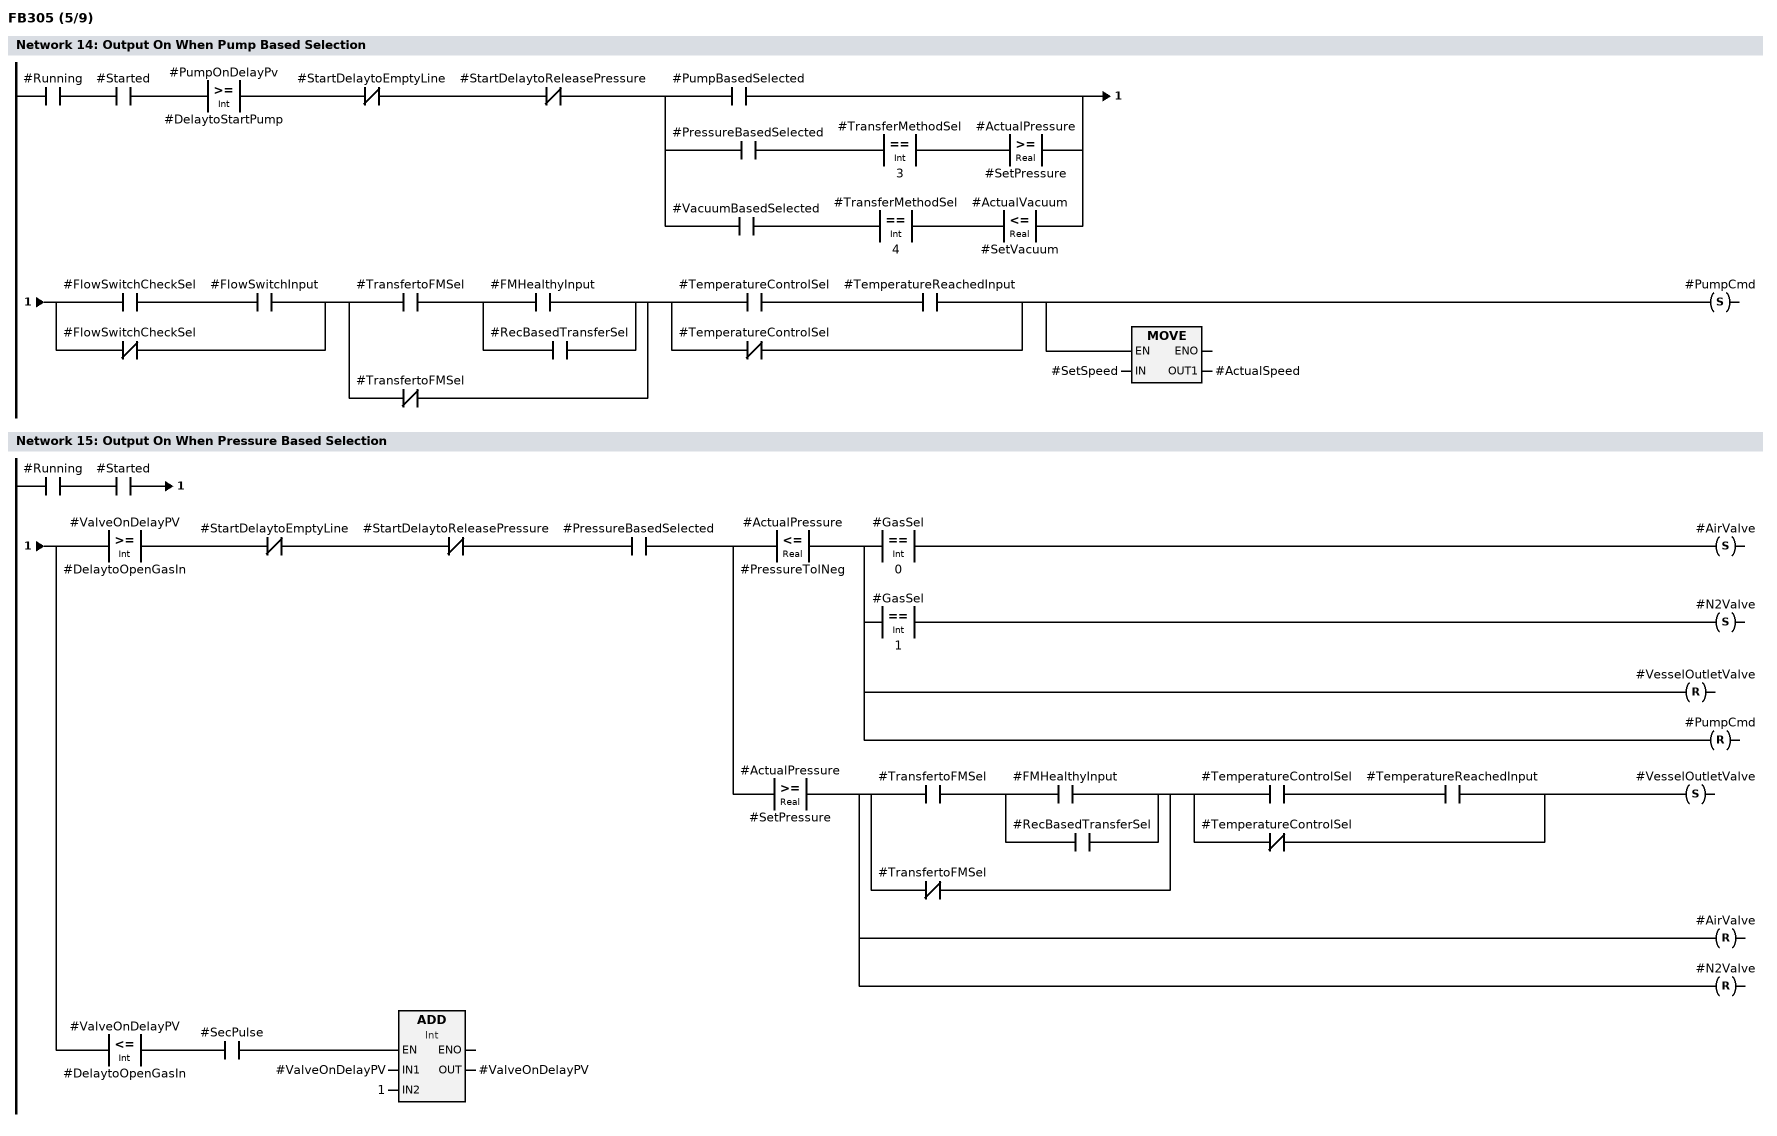
   RUNG wire#powerrail
      Contact( #Running )
      Contact( #Started )
      { S7_Templates := "SrcType := Int" } GE_Contact(in1 := #PumpOnDelayPv, in2 := #DelaytoStartPump)
      I_Contact( #StartDelaytoEmptyLine )
      I_Contact( #StartDelaytoReleasePressure )
      wire#w1
      Contact( #PumpBasedSelected )
      wire#w2
      Contact( #FlowSwitchCheckSel )
      Contact( #FlowSwitchInput )
      wire#w3
      Contact( #TransfertoFMSel )
      wire#w4
      Contact( #FMHealthyInput )
      wire#w5
      Contact( #TemperatureControlSel )
      Contact( #TemperatureReachedInput )
      wire#w6
      S_Coil( #PumpCmd )
   END_RUNG
   RUNG wire#w1
      Contact( #PressureBasedSelected )
      { S7_Templates := "SrcType := Int" } EQ_Contact(in1 := #TransferMethodSel, in2 := 3)
      { S7_Templates := "SrcType := Real" } GE_Contact(in1 := #ActualPressure, in2 := #SetPressure)
   END_RUNG wire#w2
   RUNG wire#w1
      Contact( #VacuumBasedSelected )
      { S7_Templates := "SrcType := Int" } EQ_Contact(in1 := #TransferMethodSel, in2 := 4)
      { S7_Templates := "SrcType := Real" } LE_Contact(in1 := #ActualVacuum, in2 := #SetVacuum)
   END_RUNG wire#w2
   RUNG wire#w2
      I_Contact( #FlowSwitchCheckSel )
   END_RUNG wire#w3
   RUNG wire#w4
      Contact( #RecBasedTransferSel )
   END_RUNG wire#w5
   RUNG wire#w3
      I_Contact( #TransfertoFMSel )
   END_RUNG wire#w5
   RUNG wire#w5
      I_Contact( #TemperatureControlSel )
   END_RUNG wire#w6
   RUNG wire#w6
      Move(in := #SetSpeed, out1 => #ActualSpeed)
   END_RUNG
   // the same network as SCL:
   IF #Running AND #Started AND (#PumpOnDelayPv >= #DelaytoStartPump) AND NOT #StartDelaytoEmptyLine AND NOT #StartDelaytoReleasePressure AND (#PumpBasedSelected OR (#PressureBasedSelected AND (#TransferMethodSel = 3) AND (#ActualPressure >= #SetPressure)) OR (#VacuumBasedSelected AND (#TransferMethodSel = 4) AND (#ActualVacuum <= #SetVacuum))) AND ((#FlowSwitchCheckSel AND #FlowSwitchInput) OR NOT #FlowSwitchCheckSel) AND ((#TransfertoFMSel AND (#FMHealthyInput OR #RecBasedTransferSel)) OR NOT #TransfertoFMSel) AND ((#TemperatureControlSel AND #TemperatureReachedInput) OR NOT #TemperatureControlSel) THEN
       #PumpCmd := TRUE;
       #ActualSpeed := #SetSpeed;
   END_IF;
END_REGION

REGION Network 15: Output On When Pressure Based Selection
   RUNG wire#powerrail
      Contact( #Running )
      Contact( #Started )
      wire#w1
      { S7_Templates := "SrcType := Int" } GE_Contact(in1 := #ValveOnDelayPV, in2 := #DelaytoOpenGasIn)
      I_Contact( #StartDelaytoEmptyLine )
      I_Contact( #StartDelaytoReleasePressure )
      Contact( #PressureBasedSelected )
      wire#w2
      { S7_Templates := "SrcType := Real" } LE_Contact(in1 := #ActualPressure, in2 := #PressureTolNeg)
      wire#w3
      { S7_Templates := "SrcType := Int" } EQ_Contact(in1 := #GasSel, in2 := 0)
      S_Coil( #AirValve )
   END_RUNG
   RUNG wire#w3
      { S7_Templates := "SrcType := Int" } EQ_Contact(in1 := #GasSel, in2 := 1)
      S_Coil( #N2Valve )
   END_RUNG
   RUNG wire#w3
      R_Coil( #VesselOutletValve )
   END_RUNG
   RUNG wire#w3
      R_Coil( #PumpCmd )
   END_RUNG
   RUNG wire#w2
      { S7_Templates := "SrcType := Real" } GE_Contact(in1 := #ActualPressure, in2 := #SetPressure)
      wire#w4
      Contact( #TransfertoFMSel )
      wire#w5
      Contact( #FMHealthyInput )
      wire#w6
      Contact( #TemperatureControlSel )
      Contact( #TemperatureReachedInput )
      wire#w7
      S_Coil( #VesselOutletValve )
   END_RUNG
   RUNG wire#w5
      Contact( #RecBasedTransferSel )
   END_RUNG wire#w6
   RUNG wire#w4
      I_Contact( #TransfertoFMSel )
   END_RUNG wire#w6
   RUNG wire#w6
      I_Contact( #TemperatureControlSel )
   END_RUNG wire#w7
   RUNG wire#w4
      R_Coil( #AirValve )
   END_RUNG
   RUNG wire#w4
      R_Coil( #N2Valve )
   END_RUNG
   RUNG wire#w1
      { S7_Templates := "SrcType := Int" } LE_Contact(in1 := #ValveOnDelayPV, in2 := #DelaytoOpenGasIn)
      Contact( #SecPulse )
      { S7_Templates := "SrcType := Int"; S7_GenerateENO := "TRUE" } Add(in1 := #ValveOnDelayPV, in2 := 1, out => #ValveOnDelayPV)
   END_RUNG
   // the same network as SCL:
   #_w1 := #Running AND #Started;
   #_w2 := #_w1 AND (#ValveOnDelayPV >= #DelaytoOpenGasIn) AND NOT #StartDelaytoEmptyLine AND NOT #StartDelaytoReleasePressure AND #PressureBasedSelected;
   #_w3 := #_w2 AND (#ActualPressure <= #PressureTolNeg);
   IF #_w3 AND (#GasSel = 0) THEN #AirValve := TRUE; END_IF;
   IF #_w3 AND (#GasSel = 1) THEN #N2Valve := TRUE; END_IF;
   IF #_w3 THEN
       #VesselOutletValve := FALSE;
       #PumpCmd := FALSE;
   END_IF;
   #_w4 := #_w2 AND (#ActualPressure >= #SetPressure);
   IF #_w4 AND ((#TransfertoFMSel AND (#FMHealthyInput OR #RecBasedTransferSel)) OR NOT #TransfertoFMSel) AND ((#TemperatureControlSel AND #TemperatureReachedInput) OR NOT #TemperatureControlSel) THEN
       #VesselOutletValve := TRUE;
   END_IF;
   IF #_w4 THEN
       #AirValve := FALSE;
       #N2Valve := FALSE;
   END_IF;
   IF #_w1 AND (#ValveOnDelayPV <= #DelaytoOpenGasIn) AND #SecPulse THEN
       #ValveOnDelayPV := #ValveOnDelayPV + 1;
   END_IF;
END_REGION

REGION Network 16: Output On When Vacuum Based Selection
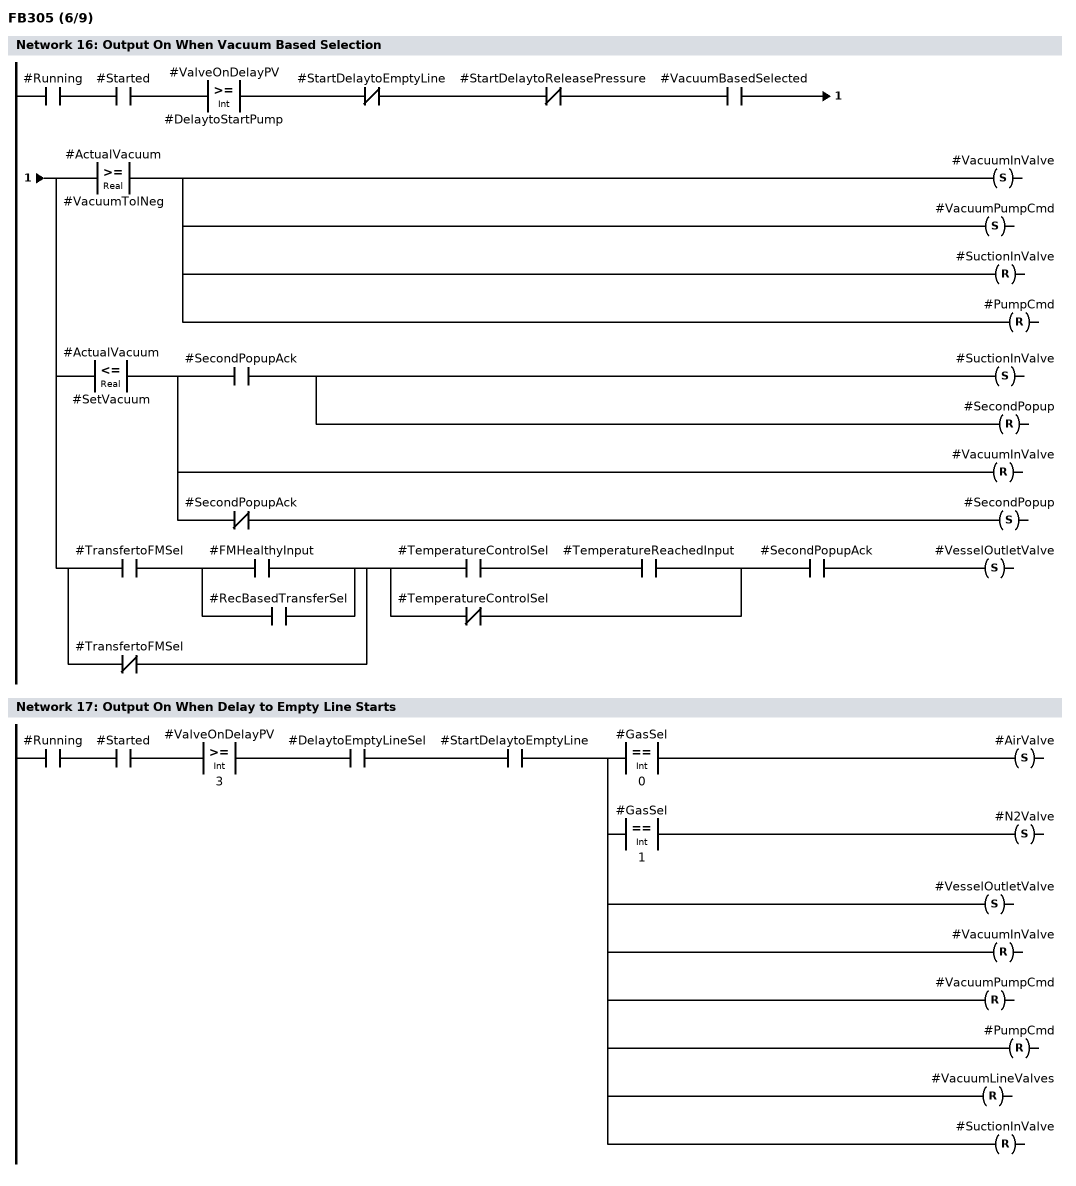
   RUNG wire#powerrail
      Contact( #Running )
      Contact( #Started )
      { S7_Templates := "SrcType := Int" } GE_Contact(in1 := #ValveOnDelayPV, in2 := #DelaytoStartPump)
      I_Contact( #StartDelaytoEmptyLine )
      I_Contact( #StartDelaytoReleasePressure )
      Contact( #VacuumBasedSelected )
      wire#w1
      { S7_Templates := "SrcType := Real" } GE_Contact(in1 := #ActualVacuum, in2 := #VacuumTolNeg)
      wire#w2
      S_Coil( #VacuumInValve )
   END_RUNG
   RUNG wire#w2
      S_Coil( #VacuumPumpCmd )
   END_RUNG
   RUNG wire#w2
      R_Coil( #SuctionInValve )
   END_RUNG
   RUNG wire#w2
      R_Coil( #PumpCmd )
   END_RUNG
   RUNG wire#w1
      { S7_Templates := "SrcType := Real" } LE_Contact(in1 := #ActualVacuum, in2 := #SetVacuum)
      wire#w3
      Contact( #SecondPopupAck )
      wire#w4
      S_Coil( #SuctionInValve )
   END_RUNG
   RUNG wire#w4
      R_Coil( #SecondPopup )
   END_RUNG
   RUNG wire#w3
      R_Coil( #VacuumInValve )
   END_RUNG
   RUNG wire#w3
      I_Contact( #SecondPopupAck )
      S_Coil( #SecondPopup )
   END_RUNG
   RUNG wire#w1
      Contact( #TransfertoFMSel )
      wire#w5
      Contact( #FMHealthyInput )
      wire#w6
      Contact( #TemperatureControlSel )
      Contact( #TemperatureReachedInput )
      wire#w7
      Contact( #SecondPopupAck )
      S_Coil( #VesselOutletValve )
   END_RUNG
   RUNG wire#w5
      Contact( #RecBasedTransferSel )
   END_RUNG wire#w6
   RUNG wire#w1
      I_Contact( #TransfertoFMSel )
   END_RUNG wire#w6
   RUNG wire#w6
      I_Contact( #TemperatureControlSel )
   END_RUNG wire#w7
   // the same network as SCL:
   #_w1 := #Running AND #Started AND (#ValveOnDelayPV >= #DelaytoStartPump) AND NOT #StartDelaytoEmptyLine AND NOT #StartDelaytoReleasePressure AND #VacuumBasedSelected;
   IF #_w1 AND (#ActualVacuum >= #VacuumTolNeg) THEN
       #VacuumInValve := TRUE;
       #VacuumPumpCmd := TRUE;
       #SuctionInValve := FALSE;
       #PumpCmd := FALSE;
   END_IF;
   #_w2 := #_w1 AND (#ActualVacuum <= #SetVacuum);
   IF #_w2 AND #SecondPopupAck THEN
       #SuctionInValve := TRUE;
       #SecondPopup := FALSE;
   END_IF;
   IF #_w2 THEN #VacuumInValve := FALSE; END_IF;
   IF #_w2 AND NOT #SecondPopupAck THEN #SecondPopup := TRUE; END_IF;
   IF #_w1 AND ((#TransfertoFMSel AND (#FMHealthyInput OR #RecBasedTransferSel)) OR NOT #TransfertoFMSel) AND ((#TemperatureControlSel AND #TemperatureReachedInput) OR NOT #TemperatureControlSel) AND #SecondPopupAck THEN
       #VesselOutletValve := TRUE;
   END_IF;
END_REGION

REGION Network 17: Output On When Delay to Empty Line Starts
   RUNG wire#powerrail
      Contact( #Running )
      Contact( #Started )
      { S7_Templates := "SrcType := Int" } GE_Contact(in1 := #ValveOnDelayPV, in2 := 3)
      Contact( #DelaytoEmptyLineSel )
      Contact( #StartDelaytoEmptyLine )
      wire#w1
      { S7_Templates := "SrcType := Int" } EQ_Contact(in1 := #GasSel, in2 := 0)
      S_Coil( #AirValve )
   END_RUNG
   RUNG wire#w1
      { S7_Templates := "SrcType := Int" } EQ_Contact(in1 := #GasSel, in2 := 1)
      S_Coil( #N2Valve )
   END_RUNG
   RUNG wire#w1
      S_Coil( #VesselOutletValve )
   END_RUNG
   RUNG wire#w1
      R_Coil( #VacuumInValve )
   END_RUNG
   RUNG wire#w1
      R_Coil( #VacuumPumpCmd )
   END_RUNG
   RUNG wire#w1
      R_Coil( #PumpCmd )
   END_RUNG
   RUNG wire#w1
      R_Coil( #VacuumLineValves )
   END_RUNG
   RUNG wire#w1
      R_Coil( #SuctionInValve )
   END_RUNG
   // the same network as SCL:
   #_w1 := #Running AND #Started AND (#ValveOnDelayPV >= 3) AND #DelaytoEmptyLineSel AND #StartDelaytoEmptyLine;
   IF #_w1 AND (#GasSel = 0) THEN #AirValve := TRUE; END_IF;
   IF #_w1 AND (#GasSel = 1) THEN #N2Valve := TRUE; END_IF;
   IF #_w1 THEN
       #VesselOutletValve := TRUE;
       #VacuumInValve := FALSE;
       #VacuumPumpCmd := FALSE;
       #PumpCmd := FALSE;
       #VacuumLineValves := FALSE;
       #SuctionInValve := FALSE;
   END_IF;
END_REGION

REGION Network 18: Output On When Pressure Release Starts
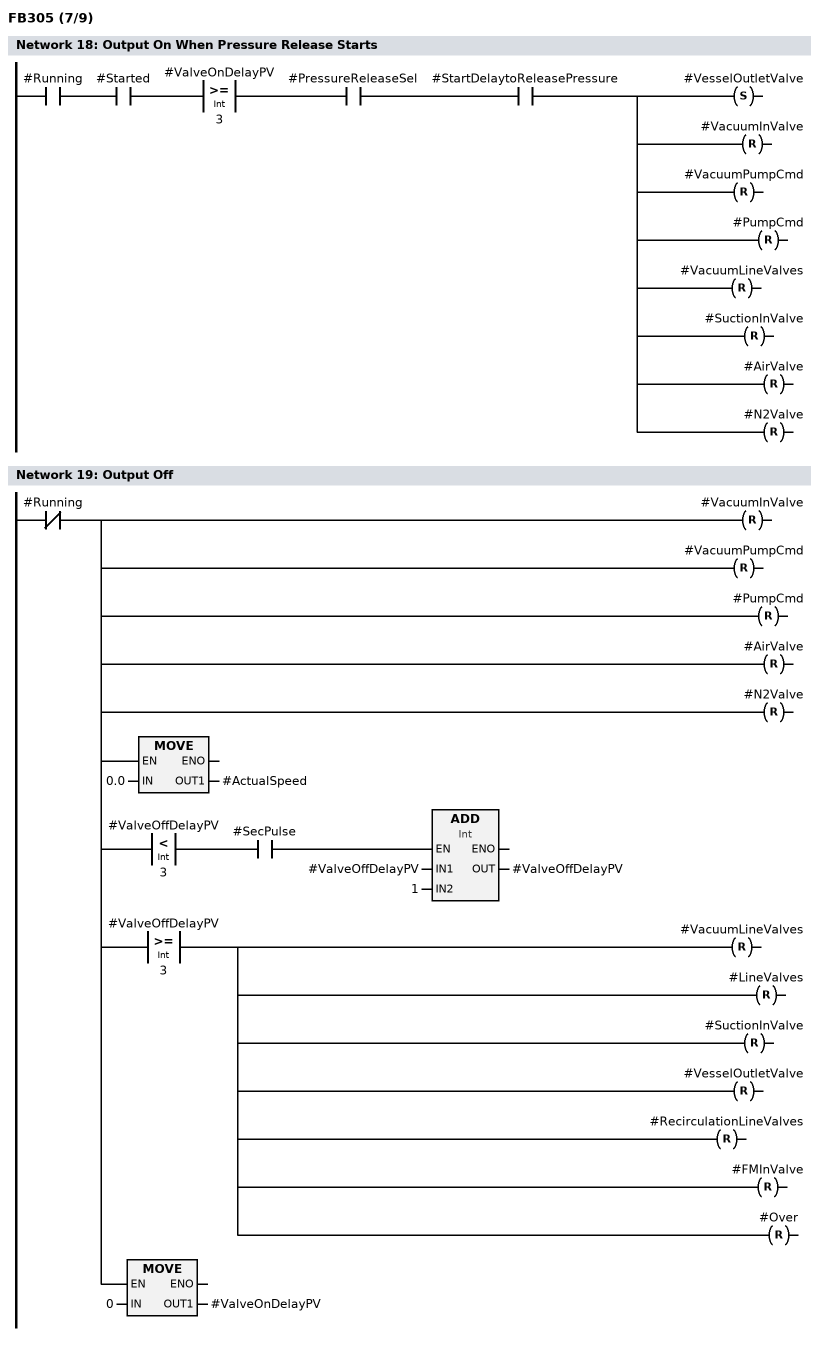
   RUNG wire#powerrail
      Contact( #Running )
      Contact( #Started )
      { S7_Templates := "SrcType := Int" } GE_Contact(in1 := #ValveOnDelayPV, in2 := 3)
      Contact( #PressureReleaseSel )
      Contact( #StartDelaytoReleasePressure )
      wire#w1
      S_Coil( #VesselOutletValve )
   END_RUNG
   RUNG wire#w1
      R_Coil( #VacuumInValve )
   END_RUNG
   RUNG wire#w1
      R_Coil( #VacuumPumpCmd )
   END_RUNG
   RUNG wire#w1
      R_Coil( #PumpCmd )
   END_RUNG
   RUNG wire#w1
      R_Coil( #VacuumLineValves )
   END_RUNG
   RUNG wire#w1
      R_Coil( #SuctionInValve )
   END_RUNG
   RUNG wire#w1
      R_Coil( #AirValve )
   END_RUNG
   RUNG wire#w1
      R_Coil( #N2Valve )
   END_RUNG
   // the same network as SCL:
   IF #Running AND #Started AND (#ValveOnDelayPV >= 3) AND #PressureReleaseSel AND #StartDelaytoReleasePressure THEN
       #VesselOutletValve := TRUE;
       #VacuumInValve := FALSE;
       #VacuumPumpCmd := FALSE;
       #PumpCmd := FALSE;
       #VacuumLineValves := FALSE;
       #SuctionInValve := FALSE;
       #AirValve := FALSE;
       #N2Valve := FALSE;
   END_IF;
END_REGION

REGION Network 19: Output Off
   RUNG wire#powerrail
      I_Contact( #Running )
      wire#w1
      R_Coil( #VacuumInValve )
   END_RUNG
   RUNG wire#w1
      R_Coil( #VacuumPumpCmd )
   END_RUNG
   RUNG wire#w1
      R_Coil( #PumpCmd )
   END_RUNG
   RUNG wire#w1
      R_Coil( #AirValve )
   END_RUNG
   RUNG wire#w1
      R_Coil( #N2Valve )
   END_RUNG
   RUNG wire#w1
      Move(in := 0.0, out1 => #ActualSpeed)
   END_RUNG
   RUNG wire#w1
      { S7_Templates := "SrcType := Int" } LT_Contact(in1 := #ValveOffDelayPV, in2 := 3)
      Contact( #SecPulse )
      { S7_Templates := "SrcType := Int"; S7_GenerateENO := "TRUE" } Add(in1 := #ValveOffDelayPV, in2 := 1, out => #ValveOffDelayPV)
   END_RUNG
   RUNG wire#w1
      { S7_Templates := "SrcType := Int" } GE_Contact(in1 := #ValveOffDelayPV, in2 := 3)
      wire#w2
      R_Coil( #VacuumLineValves )
   END_RUNG
   RUNG wire#w2
      R_Coil( #LineValves )
   END_RUNG
   RUNG wire#w2
      R_Coil( #SuctionInValve )
   END_RUNG
   RUNG wire#w2
      R_Coil( #VesselOutletValve )
   END_RUNG
   RUNG wire#w2
      R_Coil( #RecirculationLineValves )
   END_RUNG
   RUNG wire#w2
      R_Coil( #FMInValve )
   END_RUNG
   RUNG wire#w2
      R_Coil( #Over )
   END_RUNG
   RUNG wire#w1
      { S7_GenerateENO := "TRUE" } Move(in := 0, out1 => #ValveOnDelayPV)
   END_RUNG
   // the same network as SCL:
   IF NOT #Running THEN
       #VacuumInValve := FALSE;
       #VacuumPumpCmd := FALSE;
       #PumpCmd := FALSE;
       #AirValve := FALSE;
       #N2Valve := FALSE;
       #ActualSpeed := 0.0;
   END_IF;
   IF NOT #Running AND (#ValveOffDelayPV < 3) AND #SecPulse THEN
       #ValveOffDelayPV := #ValveOffDelayPV + 1;
   END_IF;
   IF NOT #Running AND (#ValveOffDelayPV >= 3) THEN
       #VacuumLineValves := FALSE;
       #LineValves := FALSE;
       #SuctionInValve := FALSE;
       #VesselOutletValve := FALSE;
       #RecirculationLineValves := FALSE;
       #FMInValve := FALSE;
       #Over := FALSE;
   END_IF;
   IF NOT #Running THEN #ValveOnDelayPV := 0; END_IF;
END_REGION

REGION Network 20: Event Status
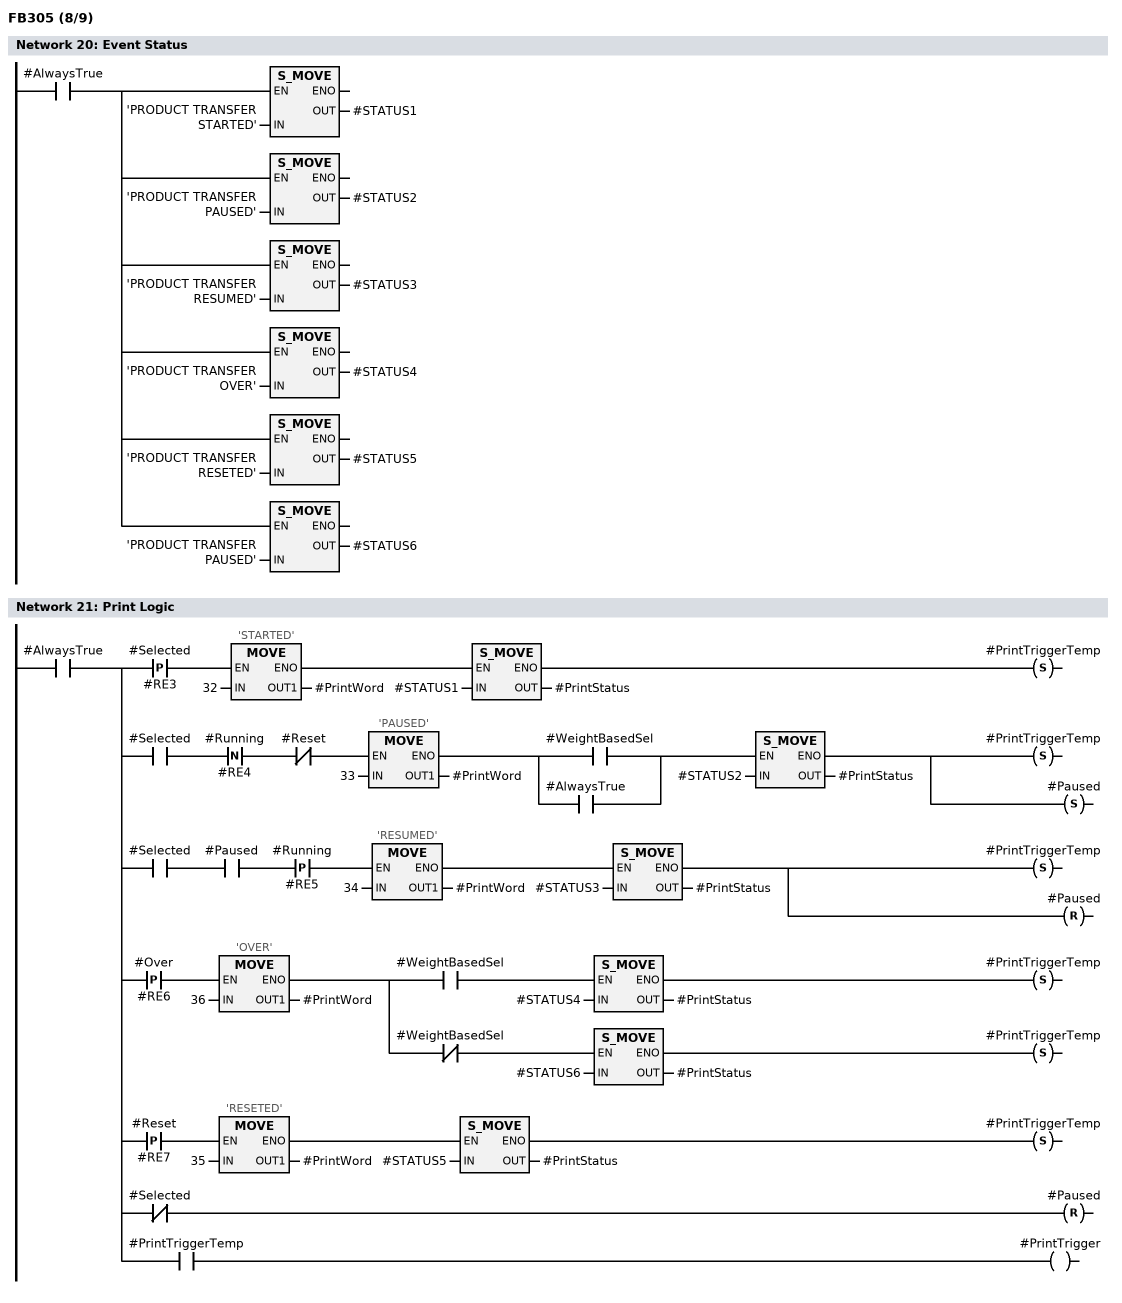
   RUNG wire#powerrail
      Contact( #AlwaysTrue )
      wire#w1
      S_Move(in := 'PRODUCT TRANSFER STARTED', out => #STATUS1)
   END_RUNG
   RUNG wire#w1
      S_Move(in := 'PRODUCT TRANSFER PAUSED', out => #STATUS2)
   END_RUNG
   RUNG wire#w1
      S_Move(in := 'PRODUCT TRANSFER RESUMED', out => #STATUS3)
   END_RUNG
   RUNG wire#w1
      S_Move(in := 'PRODUCT TRANSFER OVER', out => #STATUS4)
   END_RUNG
   RUNG wire#w1
      S_Move(in := 'PRODUCT TRANSFER RESETED', out => #STATUS5)
   END_RUNG
   RUNG wire#w1
      S_Move(in := 'PRODUCT TRANSFER PAUSED', out => #STATUS6)
   END_RUNG
   // the same network as SCL:
   IF #AlwaysTrue THEN
       #STATUS1 := 'PRODUCT TRANSFER STARTED';
       #STATUS2 := 'PRODUCT TRANSFER PAUSED';
       #STATUS3 := 'PRODUCT TRANSFER RESUMED';
       #STATUS4 := 'PRODUCT TRANSFER OVER';
       #STATUS5 := 'PRODUCT TRANSFER RESETED';
       #STATUS6 := 'PRODUCT TRANSFER PAUSED';
   END_IF;
END_REGION

REGION Network 21: Print Logic
   RUNG wire#powerrail
      Contact( #AlwaysTrue )
      wire#w1
      P_Contact(operand := #Selected, bit := #RE3)
      { S7_GenerateENO := "TRUE" } Move(in := 32, out1 => #PrintWord)   // 'STARTED'
      S_Move(in := #STATUS1, out => #PrintStatus)
      S_Coil( #PrintTriggerTemp )
   END_RUNG
   RUNG wire#w1
      Contact( #Selected )
      N_Contact(operand := #Running, bit := #RE4)
      I_Contact( #Reset )
      { S7_GenerateENO := "TRUE" } Move(in := 33, out1 => #PrintWord)   // 'PAUSED'
      wire#w2
      Contact( #WeightBasedSel )
      wire#w3
      S_Move(in := #STATUS2, out => #PrintStatus)
      wire#w4
      S_Coil( #PrintTriggerTemp )
   END_RUNG
   RUNG wire#w2
      Contact( #AlwaysTrue )
   END_RUNG wire#w3
   RUNG wire#w4
      S_Coil( #Paused )
   END_RUNG
   RUNG wire#w1
      Contact( #Selected )
      Contact( #Paused )
      P_Contact(operand := #Running, bit := #RE5)
      { S7_GenerateENO := "TRUE" } Move(in := 34, out1 => #PrintWord)   // 'RESUMED'
      S_Move(in := #STATUS3, out => #PrintStatus)
      wire#w5
      S_Coil( #PrintTriggerTemp )
   END_RUNG
   RUNG wire#w5
      R_Coil( #Paused )
   END_RUNG
   RUNG wire#w1
      P_Contact(operand := #Over, bit := #RE6)
      { S7_GenerateENO := "TRUE" } Move(in := 36, out1 => #PrintWord)   // 'OVER'
      wire#w6
      Contact( #WeightBasedSel )
      S_Move(in := #STATUS4, out => #PrintStatus)
      S_Coil( #PrintTriggerTemp )
   END_RUNG
   RUNG wire#w6
      I_Contact( #WeightBasedSel )
      S_Move(in := #STATUS6, out => #PrintStatus)
      S_Coil( #PrintTriggerTemp )
   END_RUNG
   RUNG wire#w1
      P_Contact(operand := #Reset, bit := #RE7)
      { S7_GenerateENO := "TRUE" } Move(in := 35, out1 => #PrintWord)   // 'RESETED'
      S_Move(in := #STATUS5, out => #PrintStatus)
      S_Coil( #PrintTriggerTemp )
   END_RUNG
   RUNG wire#w1
      I_Contact( #Selected )
      R_Coil( #Paused )
   END_RUNG
   RUNG wire#w1
      Contact( #PrintTriggerTemp )
      Coil( #PrintTrigger )
   END_RUNG
   // the same network as SCL:
   // ENO of a box is taken as its EN; it also drops when the box reports an error
   #_w1 := #AlwaysTrue AND #Selected AND NOT #RE3;   // rising edge of #Selected
   #RE3 := #Selected;
   IF #_w1 THEN
       #PrintWord := 32;   // 'STARTED'
       #PrintStatus := #STATUS1;
       #PrintTriggerTemp := TRUE;
   END_IF;
   #_w2 := #AlwaysTrue AND #Selected AND NOT #Running AND #RE4;   // falling edge of #Running
   #RE4 := #Running;
   #_w3 := #_w2 AND NOT #Reset;
   IF #_w3 THEN
       #PrintWord := 33;   // 'PAUSED'
   END_IF;
   IF #_w3 AND (#WeightBasedSel OR #AlwaysTrue) THEN
       #PrintStatus := #STATUS2;
       #PrintTriggerTemp := TRUE;
       #Paused := TRUE;
   END_IF;
   #_w4 := #AlwaysTrue AND #Selected AND #Paused AND #Running AND NOT #RE5;   // rising edge of #Running
   #RE5 := #Running;
   IF #_w4 THEN
       #PrintWord := 34;   // 'RESUMED'
       #PrintStatus := #STATUS3;
       #PrintTriggerTemp := TRUE;
       #Paused := FALSE;
   END_IF;
   #_w5 := #AlwaysTrue AND #Over AND NOT #RE6;   // rising edge of #Over
   #RE6 := #Over;
   IF #_w5 THEN
       #PrintWord := 36;   // 'OVER'
   END_IF;
   IF #_w5 AND #WeightBasedSel THEN
       #PrintStatus := #STATUS4;
       #PrintTriggerTemp := TRUE;
   END_IF;
   IF #_w5 AND NOT #WeightBasedSel THEN
       #PrintStatus := #STATUS6;
       #PrintTriggerTemp := TRUE;
   END_IF;
   #_w6 := #AlwaysTrue AND #Reset AND NOT #RE7;   // rising edge of #Reset
   #RE7 := #Reset;
   IF #_w6 THEN
       #PrintWord := 35;   // 'RESETED'
       #PrintStatus := #STATUS5;
       #PrintTriggerTemp := TRUE;
   END_IF;
   IF #AlwaysTrue AND NOT #Selected THEN #Paused := FALSE; END_IF;
   #PrintTrigger := #AlwaysTrue AND #PrintTriggerTemp;
END_REGION

REGION Network 22: Print Trigger Reset
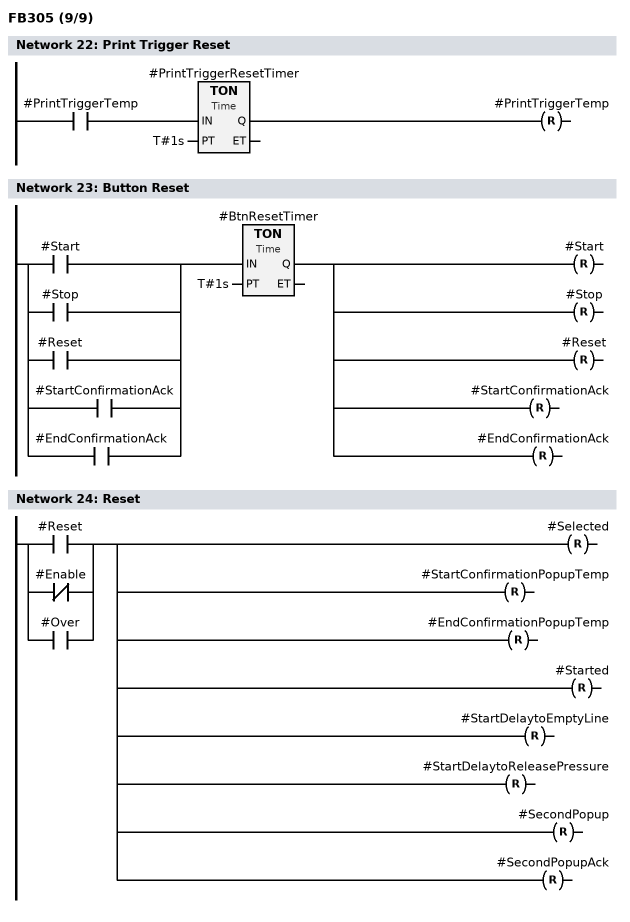
   RUNG wire#powerrail
      Contact( #PrintTriggerTemp )
      { S7_Templates := "time_type := Time" } #PrintTriggerResetTimer.TON(pt := T#1s, et =>)
      R_Coil( #PrintTriggerTemp )
   END_RUNG
   // the same network as SCL:
   #PrintTriggerResetTimer(IN := #PrintTriggerTemp, PT := T#1s);   // TON
   IF #PrintTriggerResetTimer.Q THEN #PrintTriggerTemp := FALSE; END_IF;
END_REGION

REGION Network 23: Button Reset
   RUNG wire#powerrail
      Contact( #Start )
      wire#w1
      { S7_Templates := "time_type := Time" } #BtnResetTimer.TON(pt := T#1s, et =>)
      wire#w2
      R_Coil( #Start )
   END_RUNG
   RUNG wire#powerrail
      Contact( #Stop )
   END_RUNG wire#w1
   RUNG wire#powerrail
      Contact( #Reset )
   END_RUNG wire#w1
   RUNG wire#powerrail
      Contact( #StartConfirmationAck )
   END_RUNG wire#w1
   RUNG wire#powerrail
      Contact( #EndConfirmationAck )
   END_RUNG wire#w1
   RUNG wire#w2
      R_Coil( #Stop )
   END_RUNG
   RUNG wire#w2
      R_Coil( #Reset )
   END_RUNG
   RUNG wire#w2
      R_Coil( #StartConfirmationAck )
   END_RUNG
   RUNG wire#w2
      R_Coil( #EndConfirmationAck )
   END_RUNG
   // the same network as SCL:
   #BtnResetTimer(IN := #Start OR #Stop OR #Reset OR #StartConfirmationAck OR #EndConfirmationAck, PT := T#1s);   // TON
   IF #BtnResetTimer.Q THEN
       #Start := FALSE;
       #Stop := FALSE;
       #Reset := FALSE;
       #StartConfirmationAck := FALSE;
       #EndConfirmationAck := FALSE;
   END_IF;
END_REGION

REGION Network 24: Reset
   RUNG wire#powerrail
      Contact( #Reset )
      wire#w1
      R_Coil( #Selected )
   END_RUNG
   RUNG wire#powerrail
      I_Contact( #Enable )
   END_RUNG wire#w1
   RUNG wire#powerrail
      Contact( #Over )
   END_RUNG wire#w1
   RUNG wire#w1
      R_Coil( #StartConfirmationPopupTemp )
   END_RUNG
   RUNG wire#w1
      R_Coil( #EndConfirmationPopupTemp )
   END_RUNG
   RUNG wire#w1
      R_Coil( #Started )
   END_RUNG
   RUNG wire#w1
      R_Coil( #StartDelaytoEmptyLine )
   END_RUNG
   RUNG wire#w1
      R_Coil( #StartDelaytoReleasePressure )
   END_RUNG
   RUNG wire#w1
      R_Coil( #SecondPopup )
   END_RUNG
   RUNG wire#w1
      R_Coil( #SecondPopupAck )
   END_RUNG
   // the same network as SCL:
   IF #Reset OR NOT #Enable OR #Over THEN
       #Selected := FALSE;
       #StartConfirmationPopupTemp := FALSE;
       #EndConfirmationPopupTemp := FALSE;
       #Started := FALSE;
       #StartDelaytoEmptyLine := FALSE;
       #StartDelaytoReleasePressure := FALSE;
       #SecondPopup := FALSE;
       #SecondPopupAck := FALSE;
   END_IF;
END_REGION
END_FUNCTION_BLOCK

FUNCTION_BLOCK "FB318"   // FB318, LAD
TITLE = FB318
{ S7_Optimized_Access := 'FALSE' }
AUTHOR : PRECISE
FAMILY : PRECISE
// VALVE TOGGLE
// stored: AutoNumber false, SetENOAutomatically false
   VAR_INPUT
      Enable : Bool;
      Disable : Bool;
      Fault : Bool;
      SecPulse : Bool;
      AlwaysTrue : Bool;
      StartConfirmationPopupSel : Bool;   // StartConfirmationPopupSel: 0-NO/1-YES
      EndConfirmationPopupSel : Bool;   // EndConfirmationPopupSel: 0-NO/1-YES
   END_VAR
   VAR_OUTPUT
      Valve : Bool;
      StartConfirmationPopup : Bool;   // For Start Confirmation Popup Selection: Yes
      EndConfirmationPopup : Bool;   // For End Confirmation Popup Selection: Yes
      PrintTrigger : Bool;
      PrintWord : Int;
      PrintStatus : String[50];
   END_VAR
   VAR_IN_OUT
      Open : Bool;
      Close : Bool;
      StartConfirmationAck : Bool;   // For Start Confirmation Popup Selection: Yes
      EndConfirmationAck : Bool;   // For End Confirmation Popup Selection: Yes
      SpareBtn1 : Bool;
      SpareBtn2 : Bool;
      SpareBtn3 : Bool;
      SpareBtn4 : Bool;
      Running : Bool;
      Selected : Bool;
      Over : Bool;
      StartConfirmationPopupTemp : Bool;   // For Start Confirmation Popup Selection: Yes
      EndConfirmationPopupTemp : Bool;   // For End Confirmation Popup Selection: Yes
   END_VAR
   VAR
      PrintTriggerTemp : Bool;
      RE1 : Bool;
      RE2 : Bool;
      RE3 : Bool;
      RE4 : Bool;
      RE5 : Bool;
      RE6 : Bool;
      RE7 : Bool;
      PrintTriggerResetTimer { S7_SetPoint := 'True'} : TON_TIME;
      BtnResetTimer { S7_SetPoint := 'True'} : TON_TIME;
   END_VAR
   VAR_TEMP   // added for the SCL form of the ladder/FBD networks
      _w1 : Bool;
      _w2 : Bool;
   END_VAR
BEGIN

REGION Network 1: Running
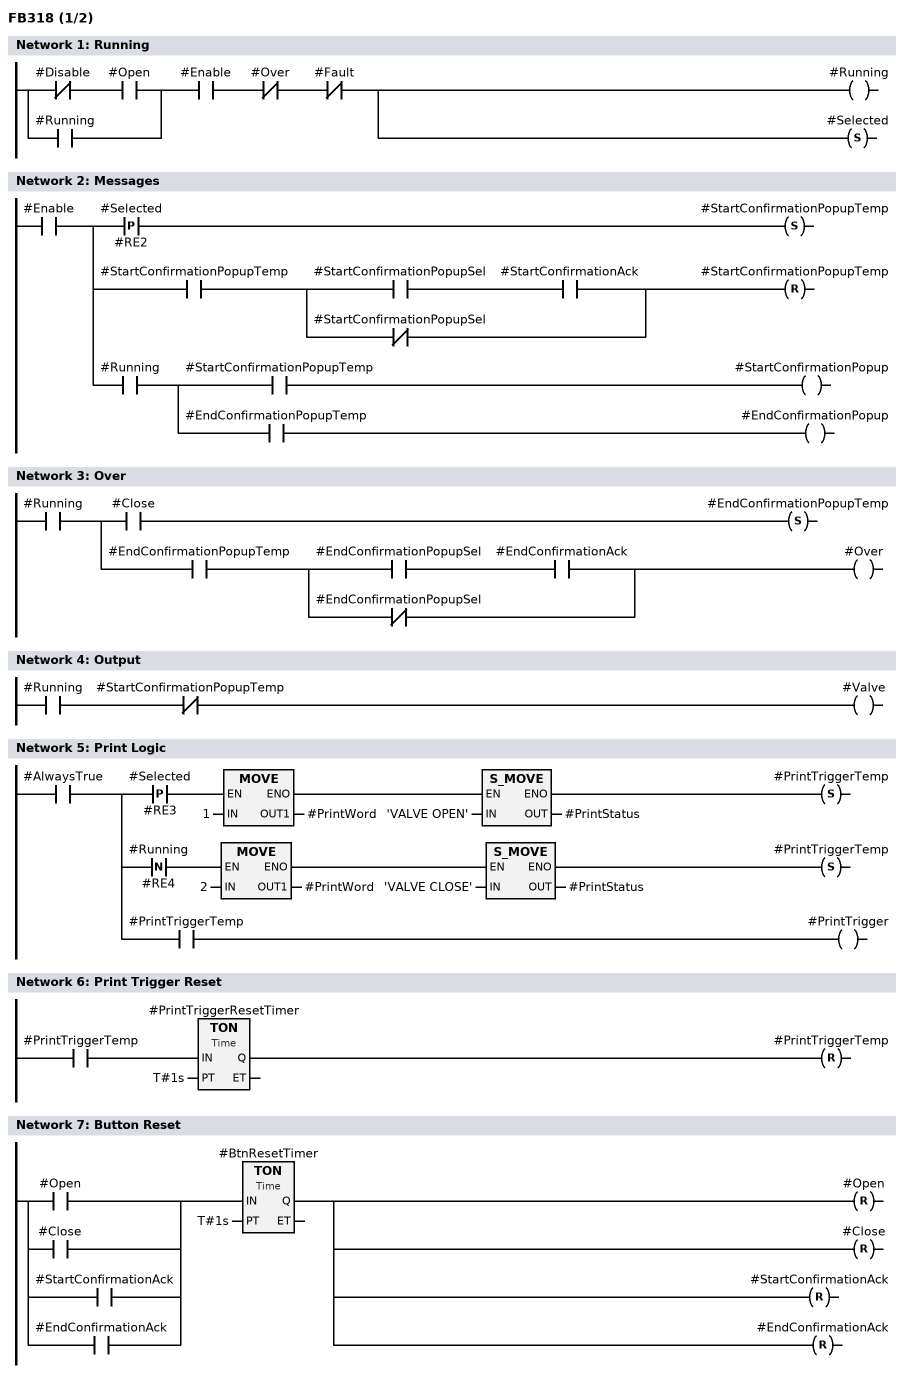
   RUNG wire#powerrail
      I_Contact( #Disable )
      Contact( #Open )
      wire#w1
      Contact( #Enable )
      I_Contact( #Over )
      I_Contact( #Fault )
      wire#w2
      Coil( #Running )
   END_RUNG
   RUNG wire#powerrail
      Contact( #Running )
   END_RUNG wire#w1
   RUNG wire#w2
      S_Coil( #Selected )
   END_RUNG
   // the same network as SCL:
   #Running := ((NOT #Disable AND #Open) OR #Running) AND #Enable AND NOT #Over AND NOT #Fault;
   IF #Running THEN #Selected := TRUE; END_IF;
END_REGION

REGION Network 2: Messages
   RUNG wire#powerrail
      Contact( #Enable )
      wire#w1
      P_Contact(operand := #Selected, bit := #RE2)
      S_Coil( #StartConfirmationPopupTemp )
   END_RUNG
   RUNG wire#w1
      Contact( #StartConfirmationPopupTemp )
      wire#w2
      Contact( #StartConfirmationPopupSel )
      Contact( #StartConfirmationAck )
      wire#w3
      R_Coil( #StartConfirmationPopupTemp )
   END_RUNG
   RUNG wire#w2
      I_Contact( #StartConfirmationPopupSel )
   END_RUNG wire#w3
   RUNG wire#w1
      Contact( #Running )
      wire#w4
      Contact( #StartConfirmationPopupTemp )
      Coil( #StartConfirmationPopup )
   END_RUNG
   RUNG wire#w4
      Contact( #EndConfirmationPopupTemp )
      Coil( #EndConfirmationPopup )
   END_RUNG
   // the same network as SCL:
   #_w1 := #Enable AND #Selected AND NOT #RE2;   // rising edge of #Selected
   #RE2 := #Selected;
   IF #_w1 THEN #StartConfirmationPopupTemp := TRUE; END_IF;
   IF #Enable AND #StartConfirmationPopupTemp AND ((#StartConfirmationPopupSel AND #StartConfirmationAck) OR NOT #StartConfirmationPopupSel) THEN
       #StartConfirmationPopupTemp := FALSE;
   END_IF;
   #_w2 := #Enable AND #Running;
   #StartConfirmationPopup := #_w2 AND #StartConfirmationPopupTemp;
   #EndConfirmationPopup := #_w2 AND #EndConfirmationPopupTemp;
END_REGION

REGION Network 3: Over
   RUNG wire#powerrail
      Contact( #Running )
      wire#w1
      Contact( #Close )
      S_Coil( #EndConfirmationPopupTemp )
   END_RUNG
   RUNG wire#w1
      Contact( #EndConfirmationPopupTemp )
      wire#w2
      Contact( #EndConfirmationPopupSel )
      Contact( #EndConfirmationAck )
      wire#w3
      Coil( #Over )
   END_RUNG
   RUNG wire#w2
      I_Contact( #EndConfirmationPopupSel )
   END_RUNG wire#w3
   // the same network as SCL:
   IF #Running AND #Close THEN #EndConfirmationPopupTemp := TRUE; END_IF;
   #Over := #Running AND #EndConfirmationPopupTemp AND ((#EndConfirmationPopupSel AND #EndConfirmationAck) OR NOT #EndConfirmationPopupSel);
END_REGION

REGION Network 4: Output
   RUNG wire#powerrail
      Contact( #Running )
      I_Contact( #StartConfirmationPopupTemp )
      Coil( #Valve )
   END_RUNG
   // the same network as SCL:
   #Valve := #Running AND NOT #StartConfirmationPopupTemp;
END_REGION

REGION Network 5: Print Logic
   RUNG wire#powerrail
      Contact( #AlwaysTrue )
      wire#w1
      P_Contact(operand := #Selected, bit := #RE3)
      { S7_GenerateENO := "TRUE" } Move(in := 1, out1 => #PrintWord)
      S_Move(in := 'VALVE OPEN', out => #PrintStatus)
      S_Coil( #PrintTriggerTemp )
   END_RUNG
   RUNG wire#w1
      N_Contact(operand := #Running, bit := #RE4)
      { S7_GenerateENO := "TRUE" } Move(in := 2, out1 => #PrintWord)
      S_Move(in := 'VALVE CLOSE', out => #PrintStatus)
      S_Coil( #PrintTriggerTemp )
   END_RUNG
   RUNG wire#w1
      Contact( #PrintTriggerTemp )
      Coil( #PrintTrigger )
   END_RUNG
   // the same network as SCL:
   // ENO of a box is taken as its EN; it also drops when the box reports an error
   #_w1 := #AlwaysTrue AND #Selected AND NOT #RE3;   // rising edge of #Selected
   #RE3 := #Selected;
   IF #_w1 THEN
       #PrintWord := 1;
       #PrintStatus := 'VALVE OPEN';
       #PrintTriggerTemp := TRUE;
   END_IF;
   #_w2 := #AlwaysTrue AND NOT #Running AND #RE4;   // falling edge of #Running
   #RE4 := #Running;
   IF #_w2 THEN
       #PrintWord := 2;
       #PrintStatus := 'VALVE CLOSE';
       #PrintTriggerTemp := TRUE;
   END_IF;
   #PrintTrigger := #AlwaysTrue AND #PrintTriggerTemp;
END_REGION

REGION Network 6: Print Trigger Reset
   RUNG wire#powerrail
      Contact( #PrintTriggerTemp )
      { S7_Templates := "time_type := Time" } #PrintTriggerResetTimer.TON(pt := T#1s, et =>)
      R_Coil( #PrintTriggerTemp )
   END_RUNG
   // the same network as SCL:
   #PrintTriggerResetTimer(IN := #PrintTriggerTemp, PT := T#1s);   // TON
   IF #PrintTriggerResetTimer.Q THEN #PrintTriggerTemp := FALSE; END_IF;
END_REGION

REGION Network 7: Button Reset
   RUNG wire#powerrail
      Contact( #Open )
      wire#w1
      { S7_Templates := "time_type := Time" } #BtnResetTimer.TON(pt := T#1s, et =>)
      wire#w2
      R_Coil( #Open )
   END_RUNG
   RUNG wire#powerrail
      Contact( #Close )
   END_RUNG wire#w1
   RUNG wire#powerrail
      Contact( #StartConfirmationAck )
   END_RUNG wire#w1
   RUNG wire#powerrail
      Contact( #EndConfirmationAck )
   END_RUNG wire#w1
   RUNG wire#w2
      R_Coil( #Close )
   END_RUNG
   RUNG wire#w2
      R_Coil( #StartConfirmationAck )
   END_RUNG
   RUNG wire#w2
      R_Coil( #EndConfirmationAck )
   END_RUNG
   // the same network as SCL:
   #BtnResetTimer(IN := #Open OR #Close OR #StartConfirmationAck OR #EndConfirmationAck, PT := T#1s);   // TON
   IF #BtnResetTimer.Q THEN
       #Open := FALSE;
       #Close := FALSE;
       #StartConfirmationAck := FALSE;
       #EndConfirmationAck := FALSE;
   END_IF;
END_REGION

REGION Network 8: Reset
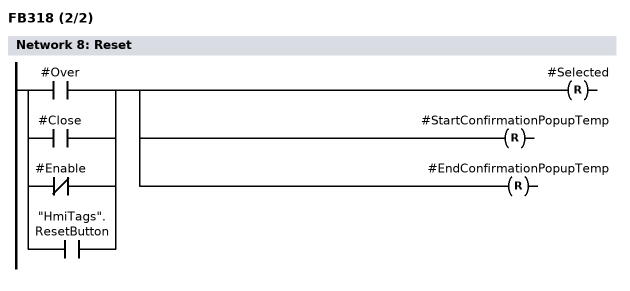
   RUNG wire#powerrail
      Contact( #Over )
      wire#w1
      R_Coil( #Selected )
   END_RUNG
   RUNG wire#powerrail
      Contact( #Close )
   END_RUNG wire#w1
   RUNG wire#powerrail
      I_Contact( #Enable )
   END_RUNG wire#w1
   RUNG wire#powerrail
      Contact( "HmiTags".ResetButton )
   END_RUNG wire#w1
   RUNG wire#w1
      R_Coil( #StartConfirmationPopupTemp )
   END_RUNG
   RUNG wire#w1
      R_Coil( #EndConfirmationPopupTemp )
   END_RUNG
   // the same network as SCL:
   IF #Over OR #Close OR NOT #Enable OR "HmiTags".ResetButton THEN
       #Selected := FALSE;
       #StartConfirmationPopupTemp := FALSE;
       #EndConfirmationPopupTemp := FALSE;
   END_IF;
END_REGION
END_FUNCTION_BLOCK

FUNCTION_BLOCK "FB317"   // FB317, LAD
TITLE = FB303
{ S7_Optimized_Access := 'FALSE' }
AUTHOR : PRECISE
FAMILY : PRECISE
// SPARGING
// stored: AutoNumber false, SetENOAutomatically false
   VAR_INPUT
      Enable : Bool;
      Disable : Bool;
      Fault : Bool;
      SecPulse : Bool;
      AlwaysTrue : Bool;
      StartConfirmationPopupSel : Bool;   // StartConfirmationPopupSel: 0-NO/1-YES
      EndConfirmationPopupSel : Bool;   // EndConfirmationPopupSel: 0-NO/1-YES
      SpargingModeSel : Int;   // Sparging Mode Selection: 0-DO/1-Time
      SpargingTimebaseSel : Bool;   // Sparging Timebase Selection: 0-sec/1-min
      SpargingLineSel : Bool;   // Sparging LineSelection: 0-THRU N2 FILTER /1-THRU VV
      N2Sel : Int;   // N2 Selection - 0-AIR/1-N2
      SetDO : Real := 10.0;   // For Sparging Mode Selection: 0-DO
      SpargingTimeMin : Int := 0;   // For Sparging Mode Selection: 1-Time & Sparging Timebase Selection: 1-min
      JdDelaySec : Int := 30;   // For Sparging Mode Selection: 1-Time & Sparging Timebase Selection: 0-sec
      PressuretoOpenVV : Real := 1.0;   // For Sparging LineSelection: 1-THRU VV
      PressuretoCloseVV : Real := 0.5;   // For Sparging LineSelection: 1-THRU VV
      ActualDO : Real;   // For Sparging Mode Selection: 0-DO
      ActualPressure : Real;   // For Sparging LineSelection: 1-THRU VV
      DelaytoOpenJd : Int := 3;
   END_VAR
   VAR_OUTPUT
      PasValve : Bool;
      N2Valve : Bool;
      JdValve : Bool;
      JvValve : Bool;   // For Sparging LineSelection: 1-THRU VV
      StartConfirmationPopup : Bool;   // For Start Confirmation Popup Selection: Yes
      EndConfirmationPopup : Bool;   // For End Confirmation Popup Selection: Yes
      SpargingTimeMinPV : DInt;
      SpargingTimeSecPV : DInt;
      PrintTrigger : Bool;
      PrintWord : Int;
      PrintStatus : String[50];
   END_VAR
   VAR_IN_OUT
      Start : Bool;
      Stop : Bool;
      Close : Bool;
      StartConfirmationAck : Bool;   // For Start Confirmation Popup Selection: Yes
      EndConfirmationAck : Bool;   // For End Confirmation Popup Selection: Yes
      SpareBtn1 : Bool;
      SpareBtn2 : Bool;
      SpareBtn3 : Bool;
      Running : Bool;
      Selected : Bool;
      Paused : Bool;
      StartConfirmationPopupTemp : Bool;   // For Start Confirmation Popup Selection: Yes
      EndConfirmationPopupTemp : Bool;   // For End Confirmation Popup Selection: Yes
      SpargingStarted : Bool;
      SpargingOver : Bool;
      SpargingTimerRunning : Bool;
   END_VAR
   VAR
      ValveOnDelayPV : Int;
      ValveOffDelayPV : Int;
      PrintTriggerTemp : Bool;
      RE1 : Bool;
      RE2 : Bool;
      RE3 : Bool;
      RE4 : Bool;
      RE5 : Bool;
      RE6 : Bool;
      RE7 : Bool;
      SpargingTimer { S7_SetPoint := 'True'} : "FB101";
      PrintTriggerResetTimer { S7_SetPoint := 'True'} : TON_TIME;
      BtnResetTimer { S7_SetPoint := 'True'} : TON_TIME;
   END_VAR
   VAR_TEMP
      STATUS1 : String[40];
      STATUS2 : String[40];
      STATUS3 : String[40];
      STATUS4 : String[40];
      STATUS5 : String[40];
   END_VAR
   VAR_TEMP   // added for the SCL form of the ladder/FBD networks
      _w1 : Bool;
      _w2 : Bool;
      _w3 : Bool;
      _w4 : Bool;
      _w5 : Bool;
   END_VAR
BEGIN

REGION Network 1: Running
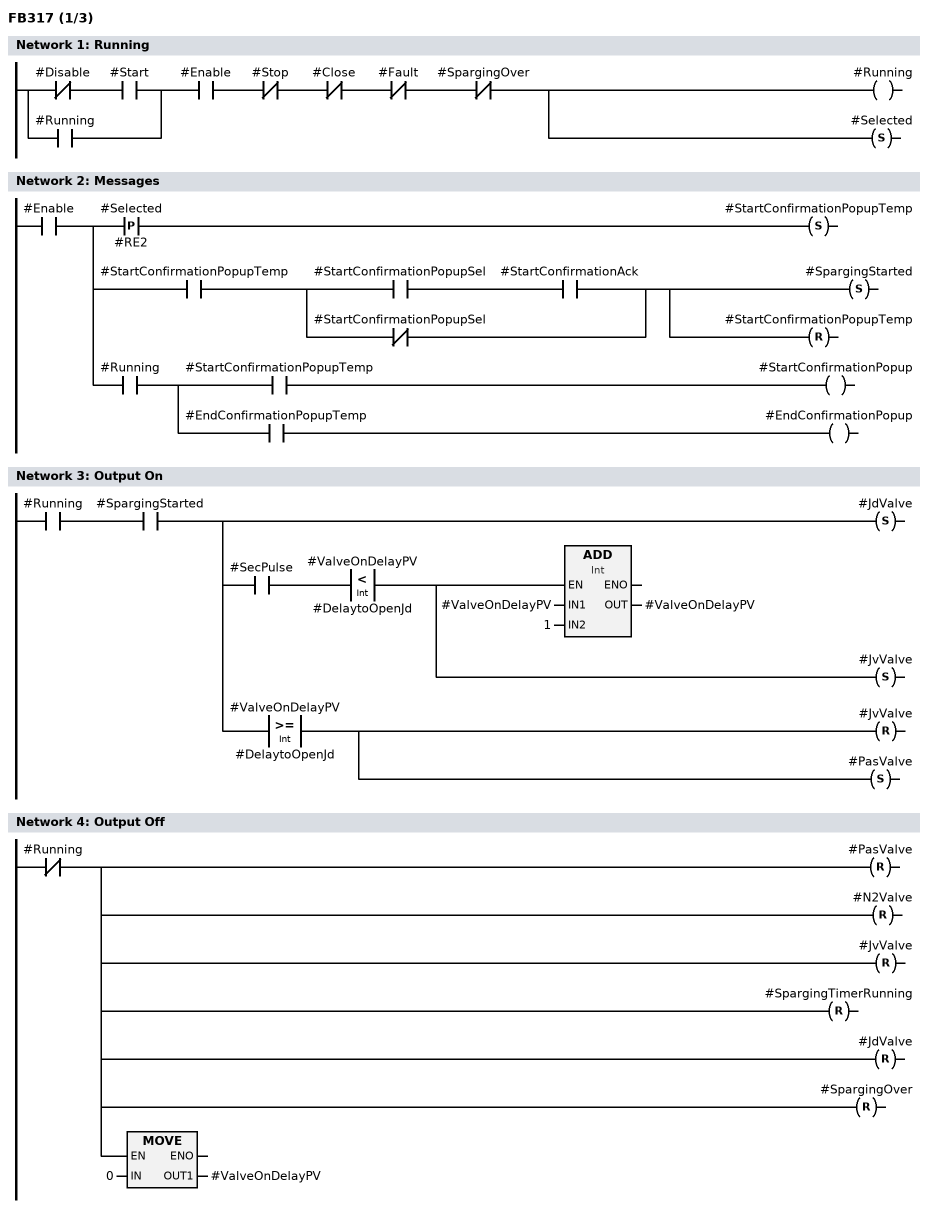
   RUNG wire#powerrail
      I_Contact( #Disable )
      Contact( #Start )
      wire#w1
      Contact( #Enable )
      I_Contact( #Stop )
      I_Contact( #Close )
      I_Contact( #Fault )
      I_Contact( #SpargingOver )
      wire#w2
      Coil( #Running )
   END_RUNG
   RUNG wire#powerrail
      Contact( #Running )
   END_RUNG wire#w1
   RUNG wire#w2
      S_Coil( #Selected )
   END_RUNG
   // the same network as SCL:
   #Running := ((NOT #Disable AND #Start) OR #Running) AND #Enable AND NOT #Stop AND NOT #Close AND NOT #Fault AND NOT #SpargingOver;
   IF #Running THEN #Selected := TRUE; END_IF;
END_REGION

REGION Network 2: Messages
   RUNG wire#powerrail
      Contact( #Enable )
      wire#w1
      P_Contact(operand := #Selected, bit := #RE2)
      S_Coil( #StartConfirmationPopupTemp )
   END_RUNG
   RUNG wire#w1
      Contact( #StartConfirmationPopupTemp )
      wire#w2
      Contact( #StartConfirmationPopupSel )
      Contact( #StartConfirmationAck )
      wire#w3
      S_Coil( #SpargingStarted )
   END_RUNG
   RUNG wire#w2
      I_Contact( #StartConfirmationPopupSel )
   END_RUNG wire#w3
   RUNG wire#w3
      R_Coil( #StartConfirmationPopupTemp )
   END_RUNG
   RUNG wire#w1
      Contact( #Running )
      wire#w4
      Contact( #StartConfirmationPopupTemp )
      Coil( #StartConfirmationPopup )
   END_RUNG
   RUNG wire#w4
      Contact( #EndConfirmationPopupTemp )
      Coil( #EndConfirmationPopup )
   END_RUNG
   // the same network as SCL:
   #_w1 := #Enable AND #Selected AND NOT #RE2;   // rising edge of #Selected
   #RE2 := #Selected;
   IF #_w1 THEN #StartConfirmationPopupTemp := TRUE; END_IF;
   IF #Enable AND #StartConfirmationPopupTemp AND ((#StartConfirmationPopupSel AND #StartConfirmationAck) OR NOT #StartConfirmationPopupSel) THEN
       #SpargingStarted := TRUE;
       #StartConfirmationPopupTemp := FALSE;
   END_IF;
   #_w2 := #Enable AND #Running;
   #StartConfirmationPopup := #_w2 AND #StartConfirmationPopupTemp;
   #EndConfirmationPopup := #_w2 AND #EndConfirmationPopupTemp;
END_REGION

REGION Network 3: Output On
   RUNG wire#powerrail
      Contact( #Running )
      Contact( #SpargingStarted )
      wire#w1
      S_Coil( #JdValve )
   END_RUNG
   RUNG wire#w1
      Contact( #SecPulse )
      { S7_Templates := "SrcType := Int" } LT_Contact(in1 := #ValveOnDelayPV, in2 := #DelaytoOpenJd)
      wire#w2
      { S7_Templates := "SrcType := Int"; S7_GenerateENO := "TRUE" } Add(in1 := #ValveOnDelayPV, in2 := 1, out => #ValveOnDelayPV)
   END_RUNG
   RUNG wire#w2
      S_Coil( #JvValve )
   END_RUNG
   RUNG wire#w1
      { S7_Templates := "SrcType := Int" } GE_Contact(in1 := #ValveOnDelayPV, in2 := #DelaytoOpenJd)
      wire#w3
      R_Coil( #JvValve )
   END_RUNG
   RUNG wire#w3
      S_Coil( #PasValve )
   END_RUNG
   // the same network as SCL:
   #_w1 := #Running AND #SpargingStarted;
   IF #_w1 THEN #JdValve := TRUE; END_IF;
   #_w2 := #_w1 AND #SecPulse AND (#ValveOnDelayPV < #DelaytoOpenJd);
   IF #_w2 THEN
       #ValveOnDelayPV := #ValveOnDelayPV + 1;
       #JvValve := TRUE;
   END_IF;
   IF #_w1 AND (#ValveOnDelayPV >= #DelaytoOpenJd) THEN
       #JvValve := FALSE;
       #PasValve := TRUE;
   END_IF;
END_REGION

REGION Network 4: Output Off
   RUNG wire#powerrail
      I_Contact( #Running )
      wire#w1
      R_Coil( #PasValve )
   END_RUNG
   RUNG wire#w1
      R_Coil( #N2Valve )
   END_RUNG
   RUNG wire#w1
      R_Coil( #JvValve )
   END_RUNG
   RUNG wire#w1
      R_Coil( #SpargingTimerRunning )
   END_RUNG
   RUNG wire#w1
      R_Coil( #JdValve )
   END_RUNG
   RUNG wire#w1
      R_Coil( #SpargingOver )
   END_RUNG
   RUNG wire#w1
      { S7_GenerateENO := "TRUE" } Move(in := 0, out1 => #ValveOnDelayPV)
   END_RUNG
   // the same network as SCL:
   IF NOT #Running THEN
       #PasValve := FALSE;
       #N2Valve := FALSE;
       #JvValve := FALSE;
       #SpargingTimerRunning := FALSE;
       #JdValve := FALSE;
       #SpargingOver := FALSE;
       #ValveOnDelayPV := 0;
   END_IF;
END_REGION

REGION Network 5: Event Status
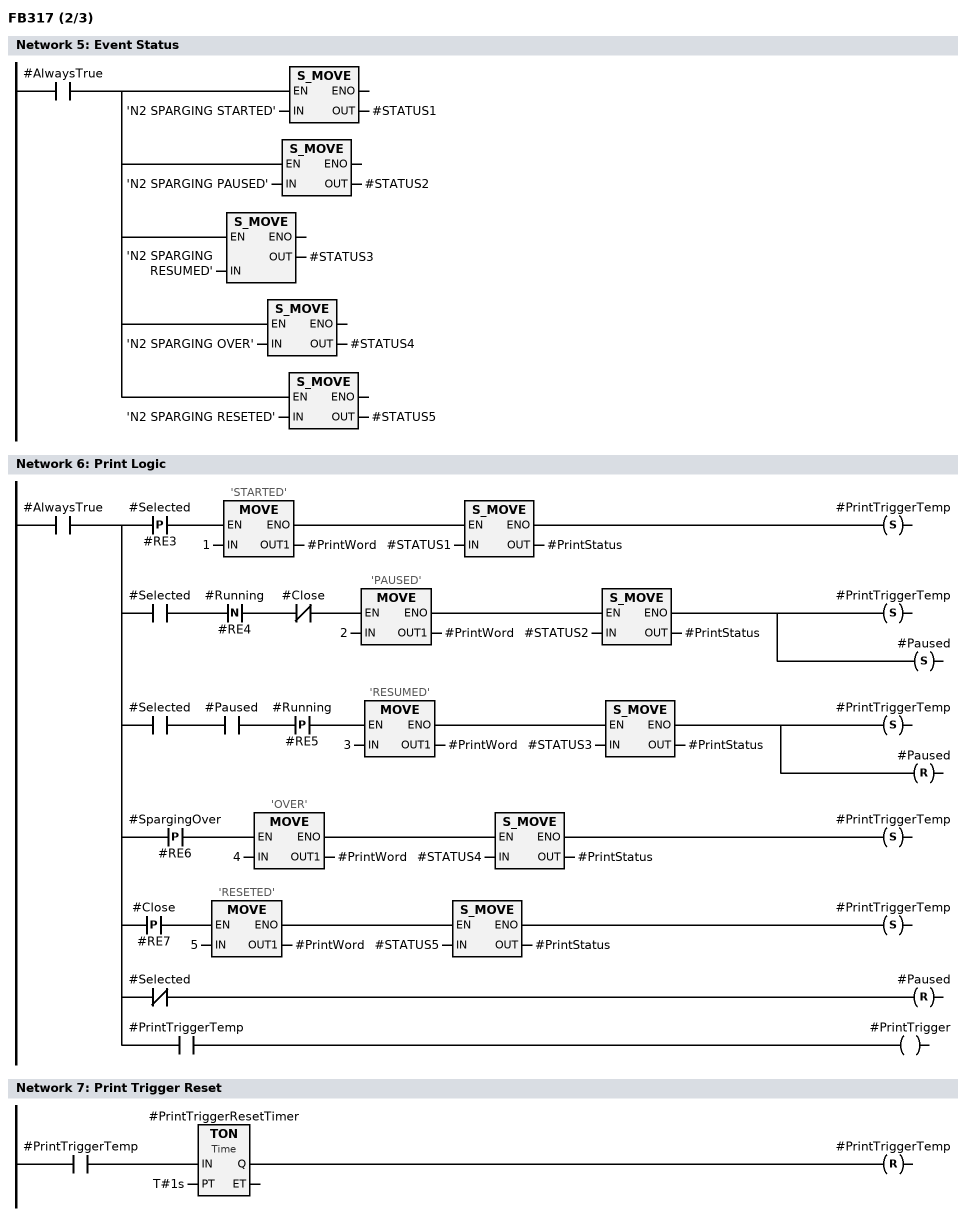
   RUNG wire#powerrail
      Contact( #AlwaysTrue )
      wire#w1
      S_Move(in := 'N2 SPARGING STARTED', out => #STATUS1)
   END_RUNG
   RUNG wire#w1
      S_Move(in := 'N2 SPARGING PAUSED', out => #STATUS2)
   END_RUNG
   RUNG wire#w1
      S_Move(in := 'N2 SPARGING RESUMED', out => #STATUS3)
   END_RUNG
   RUNG wire#w1
      S_Move(in := 'N2 SPARGING OVER', out => #STATUS4)
   END_RUNG
   RUNG wire#w1
      S_Move(in := 'N2 SPARGING RESETED', out => #STATUS5)
   END_RUNG
   // the same network as SCL:
   IF #AlwaysTrue THEN
       #STATUS1 := 'N2 SPARGING STARTED';
       #STATUS2 := 'N2 SPARGING PAUSED';
       #STATUS3 := 'N2 SPARGING RESUMED';
       #STATUS4 := 'N2 SPARGING OVER';
       #STATUS5 := 'N2 SPARGING RESETED';
   END_IF;
END_REGION

